	axis_init(
		object_name								:= CONCAT(prc_path, '_axis'), 
		axis_type								:= AXIS_TYPE_VIRTUAL, 
		encoder_scaling_factor					:= G_VIRTUAL_ENCODER_SCALING_FACTOR_DEGPINC,
		modulo									:= G_MODULO_360_DEG, 
		process									:= prc, 
		CONVERSION_this							:= axis);
	
	axis_set_max_dynamic(
		reference_velocity						:=	CONSTANTS.MAX_VELOCITY_MMpSEC,
		velocity								:=	CONSTANTS.MAX_VELOCITY_MMpSEC,
		acceleration							:=	CONSTANTS.MAX_ACCELERATION_MMpSEC2,
		deceleration							:=	CONSTANTS.MAX_DECELERATION_MMpSEC2,
		jerk									:=	CONSTANTS.MAX_JERK_MMpSEC3,
		following_error							:=	CONSTANTS.MAX_FOLLOWING_ERROR_MM,
		CONVERSION_this							:=	axis);

	jog_manager_add_axis(
		list_index					:= JOG_LIST_CSP_CASE_LOADER_VIRTUAL,
		axis						:= axis,
		master_axis					:= TRUE,
		jog_type					:= JOG_TYPE_ROTATIVE_PLUS,
		sw_limit_positive			:= 0.0,
		sw_limit_negative			:= 0.0,
		CONVERSION_this				:= csp_main_jogManager.jog_manager_virtual);
		
	boolean_init(
		object_name 							:= CONCAT(prc_path, '_case_loaded_bool'),
		process 								:= prc,
		CONVERSION_this							:= case_loaded_bool);

	check_section_asynchronous_mode_init(
		object_name:= CONCAT(prc_path, '_case_loaded_chksect'), 
		check_enable:=TRUE , 
		event_to_check:=CHECK_SECTION_EVENT_INPUT_ON , 
		execution_mode:=CHECK_SECTION_EXECUTION_WHEN_EVENT_OCCURRED , 
		diagnostic_enable:= FALSE , 
		status_bits_to_be_true:= common_global_variables.none, //ITEM_PRESENT, 
		status_bits_to_be_false:=common_global_variables.none, 
		_step_status_conditioning_execution:= FALSE, 
		status_bits_to_set:= ITEM_HAS_LOAD + ITEM_HAS_CARTON, 
		status_bits_to_reset:=common_global_variables.none , 
		reject_bit_to_set:= 0 , 
		_step:=26 , 
		first_step_to_write_offset:= 0, 
		number_of_steps_to_write:=1 , 
		reference_phase:=240 , 
		reference_phase_tolerance:= 0, 
		max_consecutive_failed_checks:= 1000000, 
		max_failed_checks_percentage:=10 , 
		products_for_failed_checks_percentage:= 10000000, 
		shift_register:= csp_case_main_statistics.sr, 
		process:= prc , 
		CONVERSION_this:= case_loaded_chksect);
		
	
			
	check_section_add_boolean_input(
			boolean_input:= case_loaded_bool,
			CONVERSION_this:= case_loaded_chksect);
		
		
	phase_init(
        object_name 				:= CONCAT(prc_path, '_load_check_ph'),
        phase 						:= 0,	//Set at runtime!
        delay 						:= 0,
        max_compensation 			:= 0,
        generator 					:= csp_main_motorization_virtualManager.phgen,
        process 					:= prc,
        CONVERSION_this 			:= load_check_ph);	
		
	phase_init(
        object_name 				:= CONCAT(prc_path, '_loader_run_check_ph'),
        phase 						:= 0,	//Set at runtime!
        delay 						:= 0,
        max_compensation 			:= 0,
        generator 					:= phgen, // CHANGE TO LOADER VIRTUAL PHGEN
        process 					:= prc,
        CONVERSION_this 			:= loader_run_check_ph);
		
	phase_generator_init(
		object_name					:= CONCAT(prc_path, '_phgen'), 
		modulo						:= axis_get_modulo(axis), 
		resolution					:= PHASE_GENERATOR_RESOLUTION_UNIT, 
		axis						:= axis, 
		process						:= prc, 
		CONVERSION_this				:= phgen);
		
		
	
	digital_check_and_message_init(
        object_name:= CONCAT(prc_path, 'product_load_failed_dchk'),
        alarm_if_input_off:= FALSE,
        alarm_delay:= 0,
        enabled_at_powerup:= TRUE,
        individual_reset:= FALSE,
        machine_reaction:=  MACHINE_REACTION_EMERGENCY_STOP,//MACHINE_REACTION_EMERGENCY_STOP,
        typology:=  MESSAGE_TYPOLOGY_ABNORMAL,//MESSAGE_TYPOLOGY_OBLIGATION,
        process:= prc,
        CONVERSION_this:= product_load_failed_dchk);
       
       
    digital_check_add_boolean(
        boolean:= product_load_failed,
        CONVERSION_this:= product_load_failed_dchk);	
		
	boolean_init(
		object_name 							:= CONCAT(prc_path, '_product_load_failed'),
		process 								:= prc,
		CONVERSION_this							:= product_load_failed);
		
		
	process_message_init(
		object_name					:=	CONCAT(prc_path, '_phase_faulted_aem'), 
		behaviour					:=	MESSAGE_BEHAVIOUR_EVENT,
		reset_timeout				:=	0,
		disableable					:=	TRUE,
		individual_reset			:=	FALSE,
		machine_reaction			:=	MACHINE_REACTION_NORMAL_STOP,
		typology					:=	MESSAGE_TYPOLOGY_ABNORMAL,
		process						:=	prc,
		CONVERSION_this				:=	phase_faulted_aem);
	
	timer_init(
		object_name					:= CONCAT(prc_path, 'phase_time_out_tmr'),
		process						:= prc,
		CONVERSION_this				:= phase_time_out_tmr);
		
	process_message_init(
		object_name					:=	CONCAT(prc_path, 'debug_immediate_stop_aem'), 
		behaviour					:=	MESSAGE_BEHAVIOUR_STATE,
		reset_timeout				:=	0,
		disableable					:=	TRUE,
		individual_reset			:=	FALSE,
		machine_reaction			:=	MACHINE_REACTION_NORMAL_STOP,
		typology					:=	MESSAGE_TYPOLOGY_ABNORMAL,
		process						:=	prc,
		CONVERSION_this				:=	debug_immediate_stop_aem);
		
	timer_init(
		object_name					:= CONCAT(prc_path, 'connection_time_out_tmr'),
		process						:= prc,
		CONVERSION_this				:= connection_time_out_tmr);
		
		
	process_message_init(
		object_name					:=	CONCAT(prc_path, '_connection_faulted_aem'), 
		behaviour					:=	MESSAGE_BEHAVIOUR_EVENT,
		reset_timeout				:=	0,
		disableable					:=	TRUE,
		individual_reset			:=	FALSE,
		machine_reaction			:=	MACHINE_REACTION_NORMAL_STOP,
		typology					:=	MESSAGE_TYPOLOGY_ABNORMAL,
		process						:=	prc,
		CONVERSION_this				:=	connection_faulted_aem);
		
	motorization_conditioner_init(
		object_name					:=	CONCAT(prc_path, 'connection_done_motcond'),
		velocity_limit				:=	0.0,
		velocity_limit_active		:=	FALSE,
		idle_handshake_active		:=	FALSE,
		execute_handshake_active	:=	TRUE,
		hold_handshake_active		:=	FALSE,
		suspend_handshake_active	:=	FALSE,
		complete_handshake_active	:=	FALSE,
		abort_handshake_active		:=	FALSE,
		stop_handshake_active		:=	FALSE,
		origin						:=	MOTORIZATION_CONDITIONER_ORIGIN_INTERNAL,
		manager						:=	csp_main_motorization_manager.motm,
		process						:=	prc,
		CONVERSION_this				:=	connection_done_motcond);
		
	process_message_init(
		object_name					:=	CONCAT(prc_path, '_Engagement_Error_aem'), 
		behaviour					:=	MESSAGE_BEHAVIOUR_EVENT,
		reset_timeout				:=	0,
		disableable					:=	TRUE,
		individual_reset			:=	FALSE,
		machine_reaction			:=	MACHINE_REACTION_EMERGENCY_STOP,
		typology					:=	MESSAGE_TYPOLOGY_ABNORMAL,
		process						:=	prc,
		CONVERSION_this				:=	Engagement_Error_aem);
		
END_IF

IF objects_running()
THEN
	motorization_conditioner_cycle(connection_done_motcond);
	phase_cycle(load_check_ph);
	phase_cycle(loader_run_check_ph);
	
	phase_generator_cycle(phgen);
	
	process_cycle(prc);
	axis_cycle(axis);
	
	digital_check_cycle(product_load_failed_dchk);
END_IF
END_ACTION

ACTION _read_process_image:
;
END_ACTION

ACTION _read_var_input:
disable_req := csp_case.disable_req;
;
END_ACTION

ACTION _set_runtime_properties:
(* Cam management *)
IF 	connection_done
THEN
	active_cam := axis.engaged_cam.cam_id;
END_IF
END_ACTION

ACTION _write_output:
;
END_ACTION

ACTION connection:
connection_conditions :=	
	NOT process_message_is_on(connection_faulted_aem)
	//AND
	//NOT jog_manager_is_jog_axis_active(JOG_LIST_CSP_CASE_VIRTUAL, csp_main_jogManager.jog_manager_virtual)
	AND
	phase_done;

(* connection_done reset *)
IF	connection_done
	AND	
	NOT connection_conditions
	AND
	NOT csp.o_machine_is_running
THEN
	connection_done := FALSE;
END_IF

(* Exit conditions *)
IF	NOT connection_conditions 
	AND
	NOT motorization_manager_is_stopping(csp_main_motorization_manager.motm)	
THEN	
	connection_status_next := CSP_CASE_STATUS_CONNECTION_ERROR;
	connection_status := connection_status_next;	
END_IF

(*************** MACHINE STATUS ***************)
CASE connection_status OF

	CSP_CASE_STATUS_CONNECTION_START:	(* Start connection *)
	
		IF	(
				motorization_manager_is_starting(csp_main_motorization_manager.motm) 
				OR
				jog_manager_is_jog_axis_active(JOG_LIST_CSP_CASE_VIRTUAL, csp_main_jogManager.jog_manager_virtual)
			)
		THEN
			connection_running := TRUE;
			connection_status_next := CSP_CASE_STATUS_CONNECTION_ENGAGE;
		END_IF
		
	CSP_CASE_STATUS_CONNECTION_ENGAGE:		
	
		master_offset_phase := csp_main_motorization_virtualManager.axis.actual_modulo_position;	
			
		axis_engage_cam(
			cam_id							:=	active_cam,	
			master_engage_mode				:=	AXIS_CAM_ENGAGE_RELATIVE,
			slave_engage_mode				:=	AXIS_CAM_ENGAGE_RELATIVE,
			activation_mode					:=	AXIS_CAM_ACTIVATION_IMMEDIATELY,
			activation_position				:=	0.0,
			master_scaling_mode				:=	AXIS_CAM_SCALING_MODE_USER_DEFINED,
			slave_scaling_mode				:=	AXIS_CAM_SCALING_MODE_AUTOOFFSET,
			master_offset					:=	LMOD(home_position_master_offset_deg + master_offset_phase, axis_get_modulo(csp_main_motorization_virtualManager.axis)),
			slave_offset					:=	0.0,
			master_scaling					:=	master_scaling,
			slave_scaling					:=	slave_scaling,
			interpolation_type				:=	AXIS_CAM_INTERPOLATION_SPLINE,	 
			master							:=	csp_main_motorization_virtualManager.axis,
			CONVERSION_this					:=	axis);
		
		connection_status_next:= CSP_TRANSFER_STATUS_CONNECTION_ENGAGED;
	
	CSP_CASE_STATUS_CONNECTION_ENGAGED:
	
		IF active_cam = 0
		THEN
			active_cam := next_cam;
		END_IF
	
		IF 	axis_is_cam_engaged(axis) 
		THEN				
			IF	active_cam <> next_cam
			THEN							
				connection_status_next := CSP_TRANSFER_STATUS_CONNECTION_CHANGE_CAM;
			ELSE
				connection_status_next:= CSP_TRANSFER_STATUS_CONNECTION_DONE;
			END_IF
		END_IF
		
	CSP_CASE_STATUS_CONNECTION_CHECK_CHANGE_CAM:						
		
		IF 	dwell
		THEN
			next_cam := DWELL_CAM;
			dwell:= FALSE;
		END_IF
				
		IF 	run
		THEN
			next_cam := FORWARD_CAM;
			run := FALSE;
		END_IF	
		
		IF	(active_cam <> next_cam)
			AND connection_conditions
		THEN							
			connection_status_next := CSP_TRANSFER_STATUS_CONNECTION_CHANGE_CAM;
		END_IF
			
		IF	NOT connection_motorization_moving
		THEN
			connection_status_next := CSP_TRANSFER_STATUS_CONNECTION_DONE;
		END_IF
			
	
	CSP_CASE_STATUS_CONNECTION_CHANGE_CAM:	
		engage_count := engage_count + 1;	
	
		axis_engage_cam(
			cam_id							:=	next_cam,	
			master_engage_mode				:=	AXIS_CAM_ENGAGE_ABSOLUTE,
			slave_engage_mode				:=	AXIS_CAM_ENGAGE_RELATIVE,
			activation_mode					:=	AXIS_CAM_ACTIVATION_NEXT_CYCLE,
			activation_position				:=	0,
			master_scaling_mode				:=	AXIS_CAM_SCALING_MODE_USER_DEFINED,
			slave_scaling_mode				:=	AXIS_CAM_SCALING_MODE_USER_DEFINED,
			master_offset					:=	home_position_master_offset_deg, 
			slave_offset					:=	0.0,
			master_scaling					:=	master_scaling,
			slave_scaling					:=	slave_scaling,
			interpolation_type				:=	AXIS_CAM_INTERPOLATION_SPLINE,	 
			master							:=	csp_main_motorization_virtualManager.axis,
			CONVERSION_this					:=	axis);	
	
		IF	motorization_manager_is_starting(csp_main_motorization_manager.motm)
		THEN
			connection_status_next := CSP_TRANSFER_STATUS_CONNECTION_DONE;
		ELSE
			IF 	axis_is_cam_engaged(axis)
			THEN
				connection_status_next := CSP_TRANSFER_STATUS_CONNECTION_WAIT_NEW_CAM;
			END_IF
		END_IF
	
	CSP_CASE_STATUS_CONNECTION_WAIT_NEW_CAM:
	
		IF	active_cam = next_cam
		THEN
			CASE next_cam OF
				DWELL_CAM:
					activation_position := next_activation_position;
				
				FORWARD_CAM:
					activation_position := 0;
					
			END_CASE
			connection_status_next := CSP_TRANSFER_STATUS_CONNECTION_CHECK_CHANGE_CAM;
		END_IF
		
		IF	NOT connection_motorization_moving
		THEN
			connection_status_next := CSP_TRANSFER_STATUS_CONNECTION_DONE;
		END_IF
		
	CSP_CASE_STATUS_CONNECTION_DONE:	(* Connection done *)	
	
		connection_running := FALSE;
		connection_done := TRUE;
		
		IF	motorization_manager_is_starting(csp_main_motorization_manager.motm)
		THEN
			motorization_conditioner_start_done(connection_done_motcond);							
			IF	active_cam <> next_cam
			THEN
				connection_status_next := CSP_TRANSFER_STATUS_CONNECTION_WAIT_NEW_CAM;
			ELSE
				connection_status_next := CSP_TRANSFER_STATUS_CONNECTION_CHECK_CHANGE_CAM;
			END_IF
		END_IF
	
	CSP_CASE_STATUS_CONNECTION_ERROR:	(* Connection error *)	
	
		IF 	connection_running
		THEN
			axis_disable(axis);
			connection_error := TRUE;						
		END_IF
		
		connection_running	:= FALSE;
		connection_done 	:= FALSE;	
		
		IF	connection_conditions
		THEN		
			connection_status_next := CSP_CASE_STATUS_CONNECTION_START;
		END_IF
		
END_CASE

IF 	NOT debug_state_machine
	OR
	debug_connection_machine_one_step	
THEN
	connection_status := connection_status_next;
	debug_connection_machine_one_step := FALSE;
END_IF

connection_motorization_moving	:= 
	motorization_manager_is_starting(csp_main_motorization_manager.motm)
	OR
	motorization_manager_is_execute(csp_main_motorization_manager.motm)
	OR
	motorization_manager_is_stopping(csp_main_motorization_manager.motm)
	OR
	motorization_manager_is_suspended(csp_main_motorization_manager.motm)
	OR
	motorization_manager_is_suspending(csp_main_motorization_manager.motm)
	OR
	motorization_manager_is_unsuspending(csp_main_motorization_manager.motm)
	OR 
	motorization_manager_is_holding(csp_main_motorization_manager.motm)
	OR
	motorization_manager_is_held(csp_main_motorization_manager.motm)
	OR
	motorization_manager_is_unholding(csp_main_motorization_manager.motm);	
	
(* Connection timeout *)
IF	(connection_running
	AND NOT debug_state_machine)	
	OR connection_error
THEN
	IF	timer_is_expired(connection_time_out_tmr)
	THEN
		process_message_set(1, connection_status, 0, connection_faulted_aem);
	END_IF
ELSE
	timer_restart(10000, connection_time_out_tmr);
END_IF
END_ACTION

ACTION phase:
phase_conditions :=
	axis_is_ok(FALSE, axis)
	AND
	process_is_ready(prc)
	AND
	process_subtree_is_ready(prc)
	//AND
	//NOT jog_manager_is_jog_axis_active(JOG_LIST_CSP_CASE_VIRTUAL, csp_main_jogManager.jog_manager_virtual)
	AND
	csp_main_motorization.motorization_axis_redefined_at_powerup
	AND
	NOT disable_req;		
	
(* phase_done reset *)
IF	phase_done
	AND
	NOT phase_conditions
	//AND 
	//NOT csp.o_machine_is_running
THEN
	//axis_disable(axis);
	phase_done:= FALSE;
END_IF

(* Exit condition *)
IF 	NOT phase_conditions
THEN
	phase_status_next := CSP_CASE_PHASE_STATUS_ERROR;
	phase_status := phase_status_next;	
END_IF

(*************** MACHINE STATUS ***************)
CASE phase_status OF

	CSP_CASE_PHASE_STATUS_START:	(* Start phasing *)
	
		IF	(
				motorization_manager_is_starting(csp_main_motorization_manager.motm) //TODOPZ: da decidere a che livello usare le variabili di i e o: wn_feeding.i_motorization_is_starting?					
				AND 
				loader_slaves_cammed
				//OR
				//jog_manager_is_jog_axis_active(JOG_LIST_CSP_CASE_VIRTUAL, csp_main_jogManager.jog_manager_virtual)
			)
		THEN
			phase_running := TRUE;			
			phase_status_next := CSP_CASE_PHASE_STATUS_DISABLE;
		END_IF
						
	CSP_CASE_PHASE_STATUS_DISABLE:
	
		axis_disable(axis);		
		
		IF 	axis_is_disabled(axis)
		THEN
			phase_status_next := CSP_CASE_PHASE_STATUS_ENABLE;
		END_IF
		
	CSP_CASE_PHASE_STATUS_ENABLE:
	
		axis_enable(axis);
		
		IF 	axis_is_enabled(axis)
		THEN
			phase_status_next := CSP_CASE_PHASE_STATUS_ENABLED;
		END_IF
		
	CSP_CASE_PHASE_STATUS_ENABLED:
	
		IF 	axis_is_standstill(axis) 
		THEN
			phase_status_next := CSP_CASE_PHASE_STATUS_CALCULATE_SLAVE_POSITION_REQUEST;								
		END_IF
		
	CSP_CASE_PHASE_STATUS_CALCULATE_SLAVE_POSITION_REQUEST:
	
		slave_position_has_been_calculated := FALSE;
	
		(* Gets the position of the master axis *)
		axis_calculate_cam_slave_master_position_deg := 
			LMOD(axis_get_actual_modulo_position(csp_main_motorization_virtualManager.axis)
			+ home_position_master_offset_deg, G_MODULO_360_DEG);
			
		(* Gets cam data for slave axis to master *)
		IF axis_calculate_cam_slave_dynamics_data(
			cam_id := active_cam,
			master_scaling := master_scaling,
			master_position := axis_calculate_cam_slave_master_position_deg,
			slave_scaling := slave_scaling,
			CONVERSION_this := axis)
		THEN
			phase_status_next := CSP_CASE_PHASE_STATUS_CALCULATING_SLAVE_POSITION;
		END_IF
	
	CSP_CASE_PHASE_STATUS_CALCULATING_SLAVE_POSITION:
	
		IF axis_cam_slave_dynamics_data_calculated(axis)
		THEN
			axis_calculated_cam_slave_position_deg := axis_get_cam_slave_dynamics_position(axis);
			slave_position_has_been_calculated := TRUE;
			phase_status_next := CSP_CASE_PHASE_STATUS_REQUEST;
				
		END_IF
		
	CSP_CASE_PHASE_STATUS_REQUEST:
		
		IF	axis_is_standstill(axis)
		THEN
			axis_move_absolute(
				position 		:= axis_calculated_cam_slave_position_deg,
				velocity 		:= phase_velocity_degps,
				direction		:= AXIS_SHORTEST_WAY,
				acceleration 	:= CONSTANTS.MOTOR_MAX_ACCELERATION_DEGPS2,
				deceleration 	:= CONSTANTS.MOTOR_MAX_DECELERATION_DEGPS2, 
				jerk 			:= CONSTANTS.MOTOR_MAX_JERK_DEGPS3, 
				buffer_mode 	:= AXIS_BUFFER_MODE_BUFFERED,
				CONVERSION_this := axis
				); 
			
		END_IF

		IF 	axis_is_absolute_moving(axis)
		THEN
			phase_status_next	:=	CSP_CASE_PHASE_STATUS_PHASING;
		END_IF

	CSP_CASE_PHASE_STATUS_PHASING:

		IF 	axis_is_standstill(axis)
		THEN
			phase_status_next	:=	CSP_TRANSFER_STATUS_PHASED;
		END_IF

	CSP_TRANSFER_STATUS_PHASED:

		IF 	engage_enable
		THEN
			phase_status_next := CSP_CASE_PHASE_STATUS_DONE;
		END_IF
		
		
	CSP_CASE_PHASE_STATUS_DONE:	(* Phase done *)	
		
		phase_running := FALSE;
		phase_done := TRUE;				
	
	CSP_CASE_PHASE_STATUS_ERROR:	(* Phase error *)
		

		IF	phase_running
		THEN
			phase_error := TRUE;
			axis_disable(axis);									
		END_IF
		phase_running := FALSE;
		
		IF	phase_conditions 	
		THEN
			phase_status_next := CSP_CASE_PHASE_STATUS_START;
		END_IF
		
END_CASE

IF 	NOT debug_state_machine
	OR
	debug_phase_machine_one_step	
THEN
	phase_status := phase_status_next;
	debug_phase_machine_one_step := FALSE;
END_IF

(* Phasing timeout *)
IF 	(phase_running
	AND NOT debug_state_machine)
	OR phase_error
THEN
	IF	timer_is_expired(phase_time_out_tmr)
	THEN
		process_message_set(1, phase_status, 0, phase_faulted_aem);
	END_IF
ELSE
	timer_restart(10000, phase_time_out_tmr);
END_IF
END_ACTION

END_PROGRAM

// ---- Application/CSP/Case/Transport/Virtual Master/csp_case_transport_virtualMaster.TcPOU
(*********************************** G.D S.p.A. - Technical Department ***********************************
============= PROGRAM INFO ============
FOLDER:             TBD
MACHINES INVOLVED:  TBD 

============= DESCRIPTION =============
csp machine declaration

============= REVISIONS ===============
Date		Version	 	Author      	Description             
----------	-------		------------  	--------------------------------------------
2019/04/05 	0000.00	 	M.Grasso		Creation of the PRG

**********************************************************************************************************)
(*$R process_ref := prc; $*)
PROGRAM csp_case_transport_virtualMaster
VAR
	
	prc:												process;
	prc_path:											STRING;
	test_pb:											BOOL:= FALSE;
	disable_pb:											BOOL:= FALSE;
	fsm_enable_condition:								BOOL := FALSE;
	fsm_next_status:									csp_case_transport_status_enum;
	fsm_status:											csp_case_transport_status_enum;
	phase_enable:										BOOL  := TRUE;
	axis: 												axis;
	phase_position_deg:									LREAL := 0;
	phase_velocity_degps:								LREAL := 20.0;
	axis_calculate_cam_slave_master_position_deg:		LREAL := 0.0;
	axis_calculated_cam_slave_position_deg:				LREAL := 0.0;
	axis_calculate_cam_master_slave_position_deg: 		LREAL := 0.0;
	axis_calculated_cam_master_position_deg: 			LREAL := 0.0;
	slave_position_has_been_calculated:					BOOL  := FALSE;
	master_position_has_been_calculated:				BOOL  := FALSE;
	engage_enable:										BOOL:=TRUE;
	target_position:									LREAL:=0;
	disable_req:										BOOL:=FALSE;
	debug_state_machine:								BOOL:=FALSE;
	debug_state_machine_one_step:						BOOL:=FALSE;
	os_minor_plow_phgen:								phase_generator;
	os_minor_plow_phwin:								phase_window;
	major_flap_phgen:									phase_generator;
	major_flap_phwin:									phase_window;
	
	transport_vm_phgen:									phase_generator;
	os_trailing_lug_pos:								LREAL;
	cam_id:												INT := LINEAR_CAM;
	slave_scaling_mm:									LREAL := 360; (*$P $*)
	master_scaling_deg:									LREAL := 360; (*$P $*)
	slave_scaling:										LREAL := 360; (*$P $*)
	master_scaling:										LREAL := 360; (*$P $*)
	home_position_master_offset_deg: 					LREAL := 0;
	running_cam:										BOOL;
	minor_plow_on: 										LREAL:=0; (*$P $*)
	minor_plow_off: 									LREAL:=100; (*$P $*)
	
	FLAG: 												STRING;
	transport_slaves_cammed:							BOOL:=FALSE;
	activation_position:    							LREAL:=0.001111;
	ls_flap_phgen:										phase_generator;
	ls_flap_on: 										LREAL := 110;
	ls_flap_off: 										LREAL := 125;
	ls_flap_phwin: 										phase_window;
	os_flap_phgen: 										phase_generator;
	os_flap_on: 										LREAL;
	os_flap_off: 										LREAL;
	os_flap_phwin: 										phase_window;
	debug: 												STRING;
	major_flap_check_on: 								LREAL:=352; (*$P $*)
	major_flap_check_off: 								LREAL:=357; (*$P $*)
	stop_for_reject: 									BOOL:=FALSE;
	PE_check: 											BOOL:=TRUE;	//initialized as true so transport virtual will run; toggle false to simulate case reject operation
	recovery_cycle:										BOOL:= FALSE;
	step_1: 											BOOL;
	step_2: 											BOOL;
	push_loader: 										BOOL;
	step_3: 											BOOL;
	step_4: 											BOOL;
	disengage_pos:										LREAL := 345;   
	latch: 												BOOL:= False;
	transport_request_latch: 							BOOL := FALSE;
	engage_after_estop: 								BOOL;
	Check_request_latch: 								BOOL := FALSE;
	Good_case_detected:									BOOL:= FALSE;
	Bad_case_detected:									BOOL:= FALSE;
	startup_follower_at_start_position:					BOOL:=FALSE;
	Startup_Good_case_detected:							BOOL := false;
	act_pos: 											LREAL := 0.995;
	reject_complete_test: 								BOOL := FALSE;
	test19:												BOOL := TRUE;
	
	PE_TEST: 											BOOL := TRUE;
	phase_done: 										BOOL := TRUE;
	Reject_again: 										BOOL := FALSE;
	pe_off: 											BOOL := TRUE;
	PE_Bypass_request:                                  BOOL:=FALSE;(*$P $*)
	consecutive_rejects_aem:							message;
	
	Abs_moved: 											BOOL;
	temp1: 												BOOL;

	Flap_control_engaged: 								BOOL;
	Reject_engaged: 									BOOL;
	Reject_disengaging: 								BOOL;
	Reject_disengaged: 									BOOL;
	Ready_to_collapse_bad_case: 						BOOL;
	Re_engaged_to_Case_Virtual: 						BOOL;
	detect_next_flaps: 									BOOL;(*$P desc:= DETECT START AND END PHASE OF FLAP EYES ON NEXT CASE; $*)
	eye_test_temp: 										BOOL;
	detected_start_phase: 								LREAL;(*$P desc:= DETECTED START PHASE OF FLAP EYES ON CASE; $*)
	detected_end_phase: 								LREAL;(*$P desc:= DETECTED END PHASE OF FLAP EYES ON CASE; $*)
	
	missing_os_fc_lower_pe_wem:							message;
	missing_os_fc_upper_pe_wem: 						message;
	missing_ls_fc_lower_pe_wem:							message;
	missing_ls_fc_upper_pe_wem: 						message;
	missing_flap: 										BOOL;
	transport_vm_ph: 									phase;
	Good_Case_For_SR: 									BOOLean;
	feed_chksect: 										check_section;
	boolean_is_resetting: 								BOOL;
	boolean_is_set: 									BOOL;
	reject_reset_boolean: 								BOOL;
	new_set: 											BOOL;
	axis_tolerance: 									INT := 30;
	phase_direction: 									BOOL;
END_VAR

VAR CONSTANT
	
	CONSTANTS:											csp_case_transport_constant_struct;

END_VAR
VAR_INPUT
	feed_reject_case_count: 							DINT;(*$M $*)
END_VAR

_read_var_input();

_object_manager();

IF NOT objects_running()
THEN
	RETURN;	
END_IF

_read_process_image();

_mode_manager();

CASE process_get_mode(prc) of
	MODE_ABSENT,
	MODE_INACTIVE:
		RETURN;
	MODE_TEST:
		_handle_process_test();
END_CASE

_set_runtime_properties();

(********************************* BODY *********************************)
				
IF  axis_is_cam_engaged(csp_case_transport_os_trailing.axis)
	AND axis_is_cam_engaged(csp_case_transport_os_leading.axis)
	AND axis_is_cam_engaged(csp_case_transport_ls_trailing.axis)
	AND axis_is_cam_engaged(csp_case_transport_ls_leading.axis)
	AND axis_is_cam_engaged(csp_case_tr_squaring_ls_leading.axis) 
	AND axis_is_cam_engaged(csp_case_tr_squaring_ls_trailing.axis)
	AND axis_is_cam_engaged(csp_case_tr_squaring_os_leading.axis)
	AND axis_is_cam_engaged(csp_case_tr_squaring_os_trailing.axis)
	AND axis_is_cam_engaged(csp_case_closing_os_horizontal.axis)
	AND axis_is_cam_engaged(csp_case_closing_os_upper.axis)
	AND axis_is_cam_engaged(csp_case_closing_os_lower.axis)
	AND axis_is_cam_engaged(csp_case_closing_ls_horizontal.axis)
	AND axis_is_cam_engaged(csp_case_closing_ls_upper.axis)
	AND axis_is_cam_engaged(csp_case_closing_ls_lower.axis)
	AND axis_is_cam_engaged(csp_case_discharge_speedbelt_ls.axis)
	AND axis_is_cam_engaged(csp_case_discharge_speedbelt_os.axis)
THEN
	transport_slaves_cammed := TRUE;
ELSE
	transport_slaves_cammed := FALSE;	
END_IF

IF axis_is_cam_engaged(csp_case_fc_os_lower_follower.axis)
	AND axis_is_cam_engaged(csp_case_fc_os_upper_follower.axis)
	AND axis_is_cam_engaged(csp_case_fc_os_lower_spreader.axis)
	AND axis_is_cam_engaged(csp_case_fc_os_upper_spreader.axis)
	AND axis_is_cam_engaged(csp_case_fc_ls_lower_follower.axis)
	AND axis_is_cam_engaged(csp_case_fc_ls_upper_follower.axis)
	AND axis_is_cam_engaged(csp_case_fc_ls_lower_spreader.axis)
	AND axis_is_cam_engaged(csp_case_fc_ls_upper_spreader.axis)
THEN
	Flap_control_engaged := TRUE;
ELSE
	Flap_control_engaged := FALSE;
END_IF



phase_window_set_phases_data(
	begin_phase:=  major_flap_check_on,
	end_phase:=  major_flap_check_off,
	begin_delay:= 0,
	end_delay:= 0,
	begin_max_compensation:= 0,
	end_max_compensation:= 0,
	CONVERSION_this:= major_flap_phwin);

IF	(
	digital_input_is_active(csp_case_fc_os_upper_sensors.flap_di)
	AND digital_input_is_active(csp_case_fc_os_lower_sensors.flap_di)
	AND digital_input_is_active(csp_case_fc_ls_upper_sensors.flap_di)
	AND digital_input_is_active(csp_case_fc_ls_lower_sensors.flap_di)
	AND NOT PE_Bypass_request
	)
	OR csp_case_main_services.dry_cycle_mode
	OR csp_main_jogManager.jog_is_active
THEN
	PE_check := TRUE;
ELSE
	Pe_check := FALSE;
END_IF

IF  ( phase_window_is_in_window(major_flap_phwin) OR (stop_for_reject AND (axis.actual_position > major_flap_check_on AND axis.actual_position < major_flap_check_off) AND axis_is_cam_engaged(axis) ))//phase_window_falling_edge(major_flap_phwin)/ 
	AND (csp_case_feed_arm_sensors.major_vacuum_sact.status = DIGITAL_ACTUATOR_STATUS_ACTIVATING OR digital_actuator_is_active(csp_case_feed_arm_sensors.major_vacuum_sact))
	AND (
		NOT PE_check
		OR NOT digital_input_is_active(csp_case_feed_arm_sensors.case_check_di)
		)
	AND csp_main_motorization_virtualManager.o_machine_is_moving 
	AND NOT csp_case_main_services.dry_cycle_mode
	AND NOT csp_case_feed_arm_sensors.mispicked_case 
THEN
	target_position := 358;
	stop_for_reject := TRUE;
	Bad_case_detected := TRUE;		
	boolean_reset(Good_Case_For_SR);
	boolean_is_resetting := TRUE;
	boolean_is_set := FALSE;
ELSIF (phase_window_is_in_window(major_flap_phwin) OR (stop_for_reject AND (axis.actual_position > major_flap_check_on AND axis.actual_position < major_flap_check_off) AND axis_is_cam_engaged(axis) ))//phase_window_falling_edge(major_flap_phwin)/ //AMR 9/1/2021
	AND PE_check
	AND (csp_case_feed_arm_sensors.major_vacuum_sact.status = DIGITAL_ACTUATOR_STATUS_ACTIVATING OR digital_actuator_is_active(csp_case_feed_arm_sensors.major_vacuum_sact))
	AND digital_input_is_active(csp_case_feed_arm_sensors.case_check_di)
	AND csp_main_motorization_virtualManager.o_machine_is_moving 
	OR csp_case_main_services.dry_cycle_mode
THEN
	boolean_set(Good_Case_For_SR);
	boolean_is_resetting := FALSE;
	boolean_is_set := TRUE;
END_IF

IF phase_edge(transport_vm_ph)//resetting at next index of shift register
THEN
	boolean_reset(Good_Case_For_SR);
END_IF

IF phase_window_falling_edge(major_flap_phwin)
	AND NOT PE_check
	AND digital_input_is_active(csp_case_feed_arm_sensors.case_check_di)
	AND NOT csp_case_main_services.dry_cycle_mode
THEN
	missing_flap := TRUE;
	ELSIF NOT digital_input_is_active(csp_case_fc_os_upper_sensors.flap_di)	AND missing_flap THEN
			process_message_set(1, 1, 1, missing_os_fc_upper_pe_wem); //message for missing fc os upper pe
	ELSIF NOT digital_input_is_active(csp_case_fc_os_lower_sensors.flap_di)	AND missing_flap THEN
			process_message_set(1, 1, 1, missing_os_fc_lower_pe_wem); //message for missing fc os lower pe
	ELSIF NOT digital_input_is_active(csp_case_fc_ls_upper_sensors.flap_di)	AND missing_flap 	THEN
			process_message_set(1, 1, 1, missing_ls_fc_upper_pe_wem); //message for missing fc ls upper pe
	ELSIF NOT digital_input_is_active(csp_case_fc_ls_lower_sensors.flap_di)	AND missing_flap 	THEN
			process_message_set(1, 1, 1, missing_ls_fc_lower_pe_wem); //message for missing fc ls lower pe
END_IF

IF(process_message_is_on(missing_os_fc_upper_pe_wem)
		OR process_message_is_on(missing_os_fc_lower_pe_wem)
		OR process_message_is_on(missing_ls_fc_upper_pe_wem)
		OR process_message_is_on(missing_ls_fc_lower_pe_wem))
		AND phase_edge(transport_vm_ph)
THEN
	process_message_reset(missing_os_fc_upper_pe_wem);
	process_message_reset(missing_os_fc_lower_pe_wem);
	process_message_reset(missing_ls_fc_upper_pe_wem);
	process_message_reset(missing_ls_fc_lower_pe_wem);
	missing_flap := FALSE;
END_IF

IF stop_for_reject
	AND csp_case_feed_virtualMaster.stop_during_reject
THEN
	stop_for_reject := FALSE;
END_IF

IF 	NOT csp_case_feed_virtualMaster.check_request
	AND csp_case_feed_virtualMaster.fsm_status <> CSP_CASE_FEED_STATUS_CAM_ENGAGED
THEN
	Bad_case_detected := FALSE;
	Good_case_detected := FALSE;
END_IF

IF csp_case_transport.transport_request 
THEN
	transport_request_latch := TRUE;
END_IF

IF transport_request_latch 
THEN
	IF axis.actual_modulo_position > 0 AND axis.actual_modulo_position < 5 OR stop_for_reject 
	THEN
		transport_request_latch := FALSE;
	END_IF
END_IF

IF 	csp_case_feed_virtualMaster.fsm_status = 157
THEN
	Startup_Good_case_detected := TRUE;
	startup_follower_at_start_position := TRUE;
ELSE
	Startup_Good_case_detected := FALSE;
	startup_follower_at_start_position := FALSE;	
END_IF

(* Turn on eye_test to capture the leading and trailing edge pe_check(when all flaps are opened successful). Use these values to then troubleshoot when eyes were lost or missed *)
IF 	detect_next_flaps
	AND NOT eye_test_temp
	AND pe_check
then
	detected_start_phase := csp_case_transport_virtualMaster.axis.actual_position;
	eye_test_temp := True;
	detect_next_flaps := False;
end_if

IF 	eye_test_temp
	AND NOT pe_check
then
	detected_end_phase := csp_case_transport_virtualMaster.axis.actual_position;
	eye_test_temp := False;
end_if

(* If stop occurs in reject operation, reset all reject bits to abort sequence and phase all axes back to starting to run *)
IF (
    machine_is_stop_emergency_active(csp.mch)
    OR machine_is_stop_normal_active(csp.mch)
    )
    AND STOP_FOR_REJECT
	OR csp_case_feed_virtualMaster.stop_during_reject
THEN
	Good_case_detected := FALSE;
	Check_request_latch :=FALSE;
	STOP_FOR_REJECT := FALSE;
	Check_request_latch :=FALSE;
	Bad_case_detected := FALSE;
	Reject_again := FALSE;
END_IF

IF (stop_for_reject 
	OR 
	reject_again)
	AND NOT temp1
THEN
	temp1 := TRUE;
	feed_reject_case_count := feed_reject_case_count + 1;
END_IF

IF 	NOT stop_for_reject 
	AND NOT reject_again
THEN
	temp1 := FALSE;
END_IF	

IF NOT csp_case_main_safety_emergency.sis.safely_closed_input.status 
	AND axis_is_cam_engaged(axis) 
THEN
	engage_after_estop := TRUE;
ELSIF csp_case_main_safety_emergency.sis.safely_closed_input.status 
	AND fsm_status = CSP_CASE_TRANSPORT_STATUS_CAM_ENGAGED 
THEN
	engage_after_estop := FALSE;
END_IF

fsm_enable_condition := axis_is_ok(FALSE, axis)
						AND
						process_is_ready(prc)
						AND
						NOT jog_manager_is_jog_axis_active(JOG_LIST_CSP_CASE_TRANSPORT_VIRTUAL, csp_main_jogManager.jog_manager_virtual)
						AND
						process_subtree_is_ready(prc)
						AND 
						NOT disable_req;
						
IF NOT fsm_enable_condition
	OR
	disable_req
	AND
	fsm_status <> CSP_CASE_TRANSPORT_STATUS_DISABLED
	AND
	fsm_status < CSP_CASE_TRANSPORT_STATUS_STOP_REQUEST
THEN
	fsm_status	:=	CSP_CASE_TRANSPORT_STATUS_STOP_REQUEST;	
END_IF

CASE fsm_status OF
	
	CSP_CASE_TRANSPORT_STATUS_NOT_INITIALIZED:
	
        IF	axis_is_ok(return_when_absent := TRUE, CONVERSION_this := axis)
        THEN
            fsm_next_status := CSP_CASE_TRANSPORT_STATUS_DISABLED;
        END_IF

		
	CSP_CASE_TRANSPORT_STATUS_DISABLED:

		IF	fsm_enable_condition
			AND
			(
				(motorization_manager_is_starting(csp_main_motorization_manager.motm))
				OR
				jog_manager_is_jog_axis_active(JOG_LIST_CSP_CASE_VIRTUAL, csp_main_jogManager.jog_manager_virtual)	
			)
		THEN
			boolean_reset(csp_case_feed_virtualMaster.case_feed_reject_active);
			fsm_next_status := CSP_CASE_TRANSPORT_STATUS_ENABLE_REQUEST;
		END_IF;

		
	CSP_CASE_TRANSPORT_STATUS_ENABLE_REQUEST:
	
		axis_enable(axis);
		IF axis_is_standstill(axis)
		THEN
	 			fsm_next_status	:=	CSP_CASE_TRANSPORT_STATUS_ENABLED;
		END_IF;		

		
	CSP_CASE_TRANSPORT_STATUS_ENABLED:


		fsm_next_status	:=	CSP_CASE_TRANSPORT_STATUS_HOME_REQUEST;

		
	CSP_CASE_TRANSPORT_STATUS_HOME_REQUEST: 

		fsm_next_status	:=	CSP_CASE_TRANSPORT_STATUS_HOME_DONE;

		
	CSP_CASE_TRANSPORT_STATUS_HOMING:

		axis.home.done := TRUE;
		IF axis_home_done(axis)
		THEN
			fsm_next_status	:=	CSP_CASE_TRANSPORT_STATUS_HOME_DONE;
		END_IF

		
	CSP_CASE_TRANSPORT_STATUS_HOME_DONE:
	
		IF phase_enable
		THEN
			fsm_next_status	:=	CSP_CASE_TRANSPORT_STATUS_CALCULATE_SLAVE_POSITION_REQUEST;
		END_IF
	
		
	CSP_CASE_TRANSPORT_STATUS_CALCULATE_SLAVE_POSITION_REQUEST:
	
		slave_position_has_been_calculated := FALSE;
		(* Gets the position of the master axis *)
		axis_calculate_cam_slave_master_position_deg := 
			LMOD(axis_get_actual_modulo_position(csp_case_virtualMaster.axis)
			+ home_position_master_offset_deg, G_MODULO_360_DEG);
		(* Gets cam data for slave axis to master *)
		IF axis_calculate_cam_slave_dynamics_data(
			cam_id := cam_id,
			master_scaling := master_scaling,
			master_position := axis_calculate_cam_slave_master_position_deg,
			slave_scaling := slave_scaling,
			CONVERSION_this := axis)
		THEN
				fsm_next_status := CSP_CASE_LOADER_STATUS_CALCULATING_SLAVE_POSITION;
		END_IF
		
		
	CSP_CASE_TRANSPORT_STATUS_CALCULATING_MASTER_POSITION:
	
		IF axis_cam_master_dynamics_data_calculated(csp_case_transport_os_trailing.axis)
		THEN
			axis_calculated_cam_master_position_deg := axis_get_cam_master_dynamics_master_axis_position_lower(axis);//csp_case_transport_os_trailing.axis
			master_position_has_been_calculated := TRUE;
			fsm_next_status := CSP_CASE_TRANSPORT_STATUS_PHASE_REQUEST;
		END_IF
		
		
	CSP_CASE_TRANSPORT_STATUS_CALCULATING_SLAVE_POSITION:
	
		IF axis_cam_slave_dynamics_data_calculated(axis)//csp_case_virtualMaster.axis
		THEN
			axis_calculated_cam_slave_position_deg := axis_get_cam_slave_dynamics_position(axis);
			slave_position_has_been_calculated := TRUE;
			fsm_next_status := CSP_CASE_TRANSPORT_STATUS_PHASE_REQUEST;
				
		END_IF
		
		
	CSP_CASE_TRANSPORT_STATUS_PHASE_REQUEST:

    	IF  LMOD((axis_calculated_cam_slave_position_deg + axis_tolerance+G_MODULO_360_DEG),G_MODULO_360_DEG)> LMOD((axis.actual_position + 360),G_MODULO_360_DEG)
        	OR
        	LMOD((axis_calculated_cam_slave_position_deg - axis_tolerance+G_MODULO_360_DEG),G_MODULO_360_DEG)< LMOD((axis.actual_position + 360),G_MODULO_360_DEG)
		THEN
			phase_direction := FALSE;    // shortest path
        ELSE
			phase_direction := TRUE; //forward
    	END_IF

		IF	axis_is_standstill(axis)(* Waits for slave axes to phase and cammed *)
			AND transport_slaves_cammed
		THEN			
			 axis_move_absolute(
				position 		:= axis_calculated_cam_slave_position_deg,
				velocity 		:= phase_velocity_degps,
				direction        := SEL(phase_direction, AXIS_SHORTEST_WAY, AXIS_POSITIVE_DIRECTION),//AXIS_SHORTEST_WAY,
				acceleration 	:= CONSTANTS.MAX_ACCELERATION_MMpSEC2/2,
				deceleration 	:= CONSTANTS.MAX_DECELERATION_MMpSEC2/2,
				jerk 			:= CONSTANTS.MAX_JERK_MMpSEC3/2, 
				buffer_mode 	:= AXIS_BUFFER_MODE_BUFFERED,
				CONVERSION_this 			:= axis
				); 
		END_IF

		IF axis_is_absolute_moving(axis)
		THEN
			fsm_next_status	:=	CSP_CASE_TRANSPORT_STATUS_PHASING;
		END_IF
	
	
	
	CSP_CASE_TRANSPORT_STATUS_PHASING:

		IF axis_is_standstill(axis)
		THEN
			phase_done := TRUE;
			fsm_next_status	:=	CSP_CASE_TRANSPORT_STATUS_PHASED;
		END_IF

		
	CSP_CASE_TRANSPORT_STATUS_PHASED:

		IF engage_enable	
		THEN
			fsm_next_status := CSP_CASE_TRANSPORT_STATUS_CAM_ENGAGED_REQ;
		END_IF


	CSP_CASE_TRANSPORT_STATUS_CAM_ENGAGED_REQ:
		 
		IF transport_slaves_cammed
		THEN	
			IF axis_get_command_velocity(csp_case_virtualMaster.axis) <1      
			THEN
				target_position :=0;
				axis_engage_cam(
					cam_id 				:= cam_id,
					master_engage_mode 	:= AXIS_CAM_ENGAGE_ABSOLUTE,
					slave_engage_mode 	:= AXIS_CAM_ENGAGE_ABSOLUTE, 
					activation_mode 	:= AXIS_CAM_ACTIVATION_IMMEDIATELY,
					activation_position	:= 0,
					master_scaling_mode	:= AXIS_CAM_SCALING_MODE_USER_DEFINED,
					slave_scaling_mode	:= AXIS_CAM_SCALING_MODE_USER_DEFINED,
					master_offset 		:= 0,
					slave_offset 		:= 0,
					master_scaling 		:= master_scaling,
					slave_scaling 		:= slave_scaling,
					interpolation_type 	:= AXIS_CAM_INTERPOLATION_SYSTEM_DEFAULT,
					master 				:= csp_case_virtualMaster.axis,
					CONVERSION_this 	:= axis);
			ELSE	
				axis_engage_cam(
					cam_id 				:= cam_id,
					master_engage_mode 	:= AXIS_CAM_ENGAGE_ABSOLUTE,
					slave_engage_mode 	:= AXIS_CAM_ENGAGE_ABSOLUTE, 
					activation_mode 	:= AXIS_CAM_ACTIVATION_AT_MASTER_CAM_POSITION,  
					activation_position	:= 0,
					master_scaling_mode	:= AXIS_CAM_SCALING_MODE_USER_DEFINED,
					slave_scaling_mode	:= AXIS_CAM_SCALING_MODE_USER_DEFINED,
					master_offset 		:= 0,
					slave_offset 		:= 0,
					master_scaling 		:= master_scaling,
					slave_scaling 		:= slave_scaling,
					interpolation_type 	:= AXIS_CAM_INTERPOLATION_SYSTEM_DEFAULT,
					master 				:= csp_case_virtualMaster.axis,
					CONVERSION_this 	:= axis);
			END_IF
		END_IF	
			
		IF	axis_is_cam_engaged(axis)
		THEN
	   		fsm_next_status := CSP_CASE_TRANSPORT_STATUS_CAM_ENGAGED;
		END_IF;
		
		
	CSP_CASE_TRANSPORT_STATUS_AXIS_ENGAGE_VERIFY :
	
		;
		
		
	CSP_CASE_TRANSPORT_STATUS_CAM_ENGAGED:
		
		IF 	NOT transport_request_latch 
			AND axis.actual_modulo_position > disengage_pos
		THEN
			fsm_next_status := CSP_CASE_TRANSPORT_STATUS_DISENGAGE_REQUEST;	
		END_IF
	
		IF NOT axis_is_enabled(axis)
		THEN
			fsm_next_status := CSP_CASE_TRANSPORT_STATUS_STOP_REQUEST;
		END_IF
	
		
	CSP_CASE_TRANSPORT_STATUS_RUNNING:

		IF motorization_manager_is_aborted(csp_main_motorization_manager.motm)
		THEN
			fsm_next_status := CSP_CASE_TRANSPORT_STATUS_STOP_REQUEST;
		END_IF
		
		
	CSP_CASE_TRANSPORT_STATUS_DISENGAGE_REQUEST:
	
		IF stop_for_reject 
		THEN
			target_position :=359.5; 
			fsm_next_status := CSP_CASE_TRANSPORT_STATUS_DISENGAGING;
		ELSE
			target_position :=0;
			fsm_next_status := CSP_CASE_TRANSPORT_STATUS_DISENGAGING;
		END_IF		
		
		
	CSP_CASE_TRANSPORT_STATUS_DISENGAGING:
	
	IF 	axis.actual_modulo_position >= disengage_pos 
		OR latch 
	THEN
		latch := TRUE;
		IF axis_disengage(
			mode:= AXIS_DISENGAGE_AND_ON_PHASE_STOP, 
			position:= target_position, 
			velocity:= 1000, 
			acceleration:= CONSTANTS.MAX_ACCELERATION_MMpSEC2, 
			deceleration:= CONSTANTS.MAX_DECELERATION_MMpSEC2, 
			jerk:= CONSTANTS.MAX_JERK_MMpSEC3, 
			CONVERSION_this:= axis)
		THEN
			IF  stop_for_reject 
			THEN
				latch := FALSE;				
				fsm_next_status := CSP_CASE_TRANSPORT_STATUS_REJECT_ABS_STEP_1;
			ELSE
				latch := FALSE;
				fsm_next_status := CSP_CASE_TRANSPORT_STATUS_CAM_ENGAGED_REQ;
			END_IF
		END_IF
	END_IF
	
	
	CSP_CASE_TRANSPORT_STATUS_STOP_REQUEST:

		axis_stop(
		    deceleration 	:= CONSTANTS.MAX_DECELERATION_MMpSEC2,
		    jerk 			:= CONSTANTS.MAX_JERK_MMpSEC3,
		    CONVERSION_this 			:= axis);

		IF 	axis_is_standstill(axis)
			OR
			NOT axis_is_ok(FALSE, axis)
			OR
			axis_is_disabled(axis)
		THEN
			fsm_next_status := CSP_CASE_TRANSPORT_STATUS_DISABLE_REQUEST;
		END_IF

		
	CSP_CASE_TRANSPORT_STATUS_DISABLE_REQUEST:
	
   		axis_disable(axis);
   		fsm_next_status := CSP_CASE_TRANSPORT_STATUS_DISABLING;

		
	CSP_CASE_TRANSPORT_STATUS_DISABLING:
	
        IF	axis_is_disabled(axis)
        THEN
            fsm_next_status := CSP_CASE_TRANSPORT_STATUS_DISABLED;
        END_IF;


	CSP_CASE_TRANSPORT_STATUS_REJECT_ABS_STEP_1:    //follower and spreaders move to zero
	
		Ready_to_collapse_bad_case := FALSE;
		
		IF stop_for_reject //AND csp_case_transport.flap_control_axes_standstill 
		THEN
			 reject_complete_test := FALSE;
			 Bad_case_detected := FALSE;
			 Reject_again := FALSE;
			 Check_request_latch := FALSE;
		END_IF
		
		IF axis_is_standstill(axis)
		THEN
			reject_complete_test := FALSE;
			Bad_case_detected := FALSE;
			Reject_again := FALSE;
			Check_request_latch := FALSE;
			axis_move_absolute(
				position 		:= csp_case_feed_virtualMaster.virtual_reject_disengage_position,
				velocity 		:= motorization_manager_get_nominal_velocity(csp_main_motorization_manager.motm),
				direction		:= AXIS_NEGATIVE_DIRECTION,
				acceleration 	:= csp_case_feed_virtualMaster.reject_accel,//CONSTANTS.MAX_ACCELERATION_MMpSEC2,
				deceleration 	:= csp_case_feed_virtualMaster.reject_accel,//CONSTANTS.MAX_DECELERATION_MMpSEC2,
				jerk 			:= CONSTANTS.MAX_JERK_MMpSEC3, 
				buffer_mode 	:= AXIS_BUFFER_MODE_BUFFERED,
				CONVERSION_this := axis); 
		END_IF
			
		IF 	axis_is_absolute_moving(axis)
		THEN
			fsm_next_status := CSP_CASE_TRANSPORT_STATUS_REJECT_ABS_STEP_2;
		END_IF
 
		
    CSP_CASE_TRANSPORT_STATUS_REJECT_ABS_STEP_2:    

		IF 	axis_is_standstill(axis) AND TRUNC(axis.actual_position) = 268
		THEN
			Ready_to_collapse_bad_case := TRUE;		
			fsm_next_status := CSP_CASE_TRANSPORT_STATUS_REJECT_ABS_STEP_3;
	 	END_IF
		
			 
	CSP_CASE_TRANSPORT_STATUS_REJECT_ABS_STEP_3:	
		
		IF csp_case_feed_virtualMaster.New_Case_Pick
		THEN	
			axis_engage_cam(
				cam_id 				:= cam_id,
				master_engage_mode 	:= AXIS_CAM_ENGAGE_ABSOLUTE,
				slave_engage_mode 	:= AXIS_CAM_ENGAGE_ABSOLUTE, 
				activation_mode 	:= AXIS_CAM_ACTIVATION_AT_MASTER_POSITION, 
				activation_position	:= csp_case_feed_virtualMaster.virtual_reject_disengage_position,
				master_scaling_mode	:= AXIS_CAM_SCALING_MODE_USER_DEFINED,
				slave_scaling_mode	:= AXIS_CAM_SCALING_MODE_AUTOOFFSET,
				master_offset 		:= 0,
				slave_offset 		:= 0,
				master_scaling 		:= master_scaling,
				slave_scaling 		:= slave_scaling,
				interpolation_type 	:= AXIS_CAM_INTERPOLATION_SYSTEM_DEFAULT,
				master 				:= csp_case_feed_virtualMaster.axis,
				CONVERSION_this 	:= axis);
		END_IF
			
		IF 	axis_is_cam_engaged(axis)
		THEN
			fsm_next_status := CSP_CASE_TRANSPORT_STATUS_REJECT_ABS_STEP_4;
		END_IF
		
		
	CSP_CASE_TRANSPORT_STATUS_REJECT_ABS_STEP_4:      

		 (* Determines if shift register will be set *)
		IF (axis.actual_position > major_flap_check_on AND axis.actual_position < major_flap_check_off) AND pe_check
			THEN 
				boolean_set(Good_Case_For_SR);
				new_set := TRUE;
		END_IF
		 
		IF 	axis_is_cam_engaged(axis) 
			AND	NOT pe_check  
			AND csp_case_feed_virtualMaster.follower_check_request							
		THEN
			Check_request_latch := FALSE;
			Bad_case_detected := TRUE;
			Reject_again := TRUE;
			process_message_set(1, 1, 1, consecutive_rejects_aem); //stop for consecutive reject 
		END_IF


        IF 	pe_check 
			AND axis_is_cam_engaged(axis)(*NOT bad_case_detected*) 
			AND csp_case_feed_virtualMaster.follower_check_request 
		THEN
			 Good_case_detected := TRUE;
			 Check_request_latch :=FALSE;
			 boolean_set(Good_Case_For_SR);
			 reject_reset_boolean := TRUE;
			 STOP_FOR_REJECT := FALSE;
			 Re_engaged_to_Case_Virtual := FALSE;
			 fsm_next_status := CSP_CASE_TRANSPORT_STATUS_RECOVERY_CAM_ENGAGED_REQ;
         END_IF
	
		
	CSP_CASE_TRANSPORT_STATUS_RECOVERY_CAM_ENGAGED_REQ:
		
		IF 	axis_is_cam_engaged(axis) 
			AND NOT Re_engaged_to_Case_Virtual
		THEN
			axis_disengage(
				mode:= AXIS_DISENGAGE_AND_STOP, 
				position 		:= 0,
				velocity:= 1000, 
				acceleration:= CONSTANTS.MAX_ACCELERATION_MMpSEC2, 
				deceleration:= CONSTANTS.MAX_DECELERATION_MMpSEC2, 
				jerk:= CONSTANTS.MAX_JERK_MMpSEC3, 
				CONVERSION_this 			:= axis ); 
			Reject_disengaging := TRUE;
		END_IF
		
		IF 	Reject_disengaging 
			AND axis_is_disengaged(axis)
		THEN
			Reject_disengaged := TRUE;
		END_IF
		

	IF 	csp_case_feed.feed_request
		AND axis_is_standstill(axis)
		AND TRUNC(axis.actual_position) = 0
		AND Reject_disengaged
	THEN
		
		axis_engage_cam(
				cam_id 				:= cam_id,
				master_engage_mode 	:= AXIS_CAM_ENGAGE_ABSOLUTE,
				slave_engage_mode 	:= AXIS_CAM_ENGAGE_ABSOLUTE, 
				activation_mode 	:= AXIS_CAM_ACTIVATION_IMMEDIATELY, 
				activation_position	:= 0,
				master_scaling_mode	:= AXIS_CAM_SCALING_MODE_USER_DEFINED,
				slave_scaling_mode	:= AXIS_CAM_SCALING_MODE_USER_DEFINED,
				master_offset 		:= 0,
				slave_offset 		:= 0,
				master_scaling 		:= master_scaling,
				slave_scaling 		:= slave_scaling,
				interpolation_type 	:= AXIS_CAM_INTERPOLATION_SYSTEM_DEFAULT,
				master 				:= csp_case_virtualMaster.axis,
				CONVERSION_this 	:= axis);	
		Re_engaged_to_Case_Virtual := TRUE;
	END_IF			
		
	IF 	axis_is_cam_engaged(axis) 
		AND Re_engaged_to_Case_Virtual 
	THEN
		step_4:= FALSE;
		Abs_moved := FALSE; //Resets bit for reject again
		reject_complete_test := TRUE;
		Good_case_detected := FALSE;
		Reject_disengaged := FALSE;
		Reject_disengaging := FALSE;
		fsm_next_status := CSP_CASE_TRANSPORT_STATUS_CAM_ENGAGED;
	
		IF pe_check (*NOT bad_case_detected*) 
			AND Stop_for_reject
			AND axis_is_cam_engaged(csp_case_fc_os_lower_follower.axis)
			AND axis_is_cam_engaged(csp_case_fc_os_upper_follower.axis)
			AND axis_is_cam_engaged(csp_case_fc_ls_lower_follower.axis)
			AND axis_is_cam_engaged(csp_case_fc_ls_upper_follower.axis)
			AND csp_case_transport.Spreaders_Extended
			AND axis_is_cam_engaged(csp_case_feed_virtualMaster.axis)	
		THEN
			STOP_FOR_REJECT := FALSE;
		END_IF
	END_IF
		
END_CASE;

IF NOT debug_state_machine
	OR
	debug_state_machine_one_step
THEN
	fsm_status := fsm_next_status;
	debug_state_machine_one_step := FALSE;
END_IF

(************************************************************************)

_handle_messages();

_write_output();

ACTION _handle_messages:
IF (
	machine_is_stopped(csp.mch)
	OR machine_is_stop_emergency_active(csp.mch)
	)
	AND process_message_is_on(consecutive_rejects_aem)
THEN
	bad_case_detected := FALSE;
	Good_case_detected := FALSE;
	process_message_reset(consecutive_rejects_aem);
		
END_IF;
END_ACTION

ACTION _handle_process_test:
;
END_ACTION

ACTION _mode_manager:
IF process_mode_req_is_pending(prc)
THEN
    process_apply_mode_req_first_step(prc);
    CASE process_get_mode(prc) OF
        MODE_TO_ABSENT:
			;
        MODE_TO_INACTIVE:
			;
        MODE_TO_TEST:
			;
        MODE_TO_OPERATIONAL:
			;
    END_CASE
    process_apply_mode_req_second_step(prc);
END_IF
END_ACTION

ACTION _object_manager:
IF objects_initialization()
THEN
	sub_process_init(
		object_name								:= 'csp_case_transport_virtualMaster.prc', 
		process									:= csp_case_transport.prc, 
		CONVERSION_this							:= prc);
		
	prc_path 									:= process_get_path(prc);
	
	axis_init(
		object_name								:= CONCAT(prc_path, '_axis'), 
		axis_type								:= AXIS_TYPE_VIRTUAL, 
		encoder_scaling_factor					:= G_VIRTUAL_ENCODER_SCALING_FACTOR_DEGPINC,
		modulo									:= G_MODULO_360_DEG, 
		process									:= prc, 
		CONVERSION_this							:= axis);
	
	axis_set_max_dynamic(
		reference_velocity						:=	CONSTANTS.MAX_VELOCITY_MMpSEC,
		velocity								:=	CONSTANTS.MAX_VELOCITY_MMpSEC,
		acceleration							:=	CONSTANTS.MAX_ACCELERATION_MMpSEC2,
		deceleration							:=	CONSTANTS.MAX_DECELERATION_MMpSEC2,
		jerk									:=	CONSTANTS.MAX_JERK_MMpSEC3,
		following_error							:=	CONSTANTS.MAX_FOLLOWING_ERROR_MM,
		CONVERSION_this							:=	axis);
		
	jog_manager_add_axis(
		list_index								:= JOG_LIST_CSP_CASE_TRANSPORT_VIRTUAL,
		axis									:= axis,
		master_axis								:= TRUE,
		jog_type								:= JOG_TYPE_ROTATIVE_PLUS,
		sw_limit_positive						:= 0.0,
		sw_limit_negative						:= 0.0,
		CONVERSION_this							:= csp_main_jogManager.jog_manager_virtual);

//Created to be the axis for the shift registers	
	phase_generator_init(
		object_name								:=CONCAT(PRC_PATH, '_transport_vm_phgen'), 
		modulo									:=360 , 
		resolution								:= PHASE_GENERATOR_RESOLUTION_UNIT, 
		axis									:=axis, 
		process									:=prc , 
		CONVERSION_this							:= transport_vm_phgen);
//Upper major flap check cam and phase generator	

//Lower major flap check cam and phase generator		
	
	phase_window_init(
		object_name								:=CONCAT(PRC_PATH, '_major_lower_flap_phwin'), 
		begin_phase								:=major_flap_check_on, 
		end_phase								:=major_flap_check_off, 
		begin_delay								:=0, 
		end_delay								:=0, 
		begin_max_compensation					:=0, 
		end_max_compensation					:=0, 
		generator								:=transport_vm_phgen , 
		process									:=prc , 
		CONVERSION_this							:=major_flap_phwin);	

//OS minor plow cam window and phase generator
	
	phase_window_init(
		object_name								:=CONCAT(PRC_PATH, '_os_minor_plow_phwin'), 
		begin_phase								:=minor_plow_on, 
		end_phase								:=minor_plow_off, 
		begin_delay								:=0, 
		end_delay								:=0, 
		begin_max_compensation					:=0, 
		end_max_compensation					:=0, 
		generator								:=transport_vm_phgen , 
		process									:=prc , 
		CONVERSION_this							:=os_minor_plow_phwin);	



//LS open flap cam window and phase generator
	
	
	phase_window_init(
		object_name								:=CONCAT(PRC_PATH, '_ls_flap_phwin'), 
		begin_phase								:=ls_flap_on, 
		end_phase								:=ls_flap_off, 
		begin_delay								:=0, 
		end_delay								:=0, 
		begin_max_compensation					:=0, 
		end_max_compensation					:=0, 
		generator								:=transport_vm_phgen , 
		process									:=prc , 
		CONVERSION_this							:=ls_flap_phwin);	

//OS open flap cam window and phase generator		
	
	phase_window_init(
		object_name								:=CONCAT(PRC_PATH, '_os_flap_phwin'), 
		begin_phase								:=os_flap_on, 
		end_phase								:=os_flap_off, 
		begin_delay								:=0, 
		end_delay								:=0, 
		begin_max_compensation					:=0, 
		end_max_compensation					:=0, 
		generator								:=transport_vm_phgen , 
		process									:=prc , 
		CONVERSION_this							:=os_flap_phwin);
		
//transport vm phase edge		
	 phase_init(
        object_name               				:= CONCAT(prc_path, '_transport_vm_ph'),
        phase                         			:= 0,    //Set at runtime!
        delay                         			:= 0,
        max_compensation             			:= 0,
        generator                    			:= transport_vm_phgen, 
        process                     			:= prc,
        CONVERSION_this             			:= transport_vm_ph);

		
		process_message_init(
		object_name:= CONCAT(prc_path, '_consecutive_reject_aem'), 
		behaviour:= MESSAGE_BEHAVIOUR_STATE, 
		reset_timeout:= 0, 
		disableable:= FALSE, 
		individual_reset:= FALSE, 
		machine_reaction:= MACHINE_REACTION_STOP_IN_PHASE_ONE, 
		typology:= MESSAGE_TYPOLOGY_ABNORMAL, 
		process:= prc, 
		CONVERSION_this:= consecutive_rejects_aem);
		
		process_message_init(
        object_name:= CONCAT(prc_path, '_missing_os_fc_lower_pe_wem'),
        behaviour:= MESSAGE_BEHAVIOUR_EVENT,
        reset_timeout:= 0,
        disableable:= TRUE,
        individual_reset:= FALSE,
        machine_reaction:= MACHINE_REACTION_NO_STOP,
        typology:=  MESSAGE_TYPOLOGY_NORMAL,
        process:= prc,
        CONVERSION_this:= missing_os_fc_lower_pe_wem);       
       
       
        process_message_init(
        object_name:= CONCAT(prc_path, '_missing_os_fc_upper_pe_wem'),
        behaviour:= MESSAGE_BEHAVIOUR_EVENT,
        reset_timeout:= 0,
        disableable:= TRUE,
        individual_reset:= FALSE,
        machine_reaction:= MACHINE_REACTION_NO_STOP,
        typology:=  MESSAGE_TYPOLOGY_NORMAL,
        process:= prc,
        CONVERSION_this:= missing_os_fc_upper_pe_wem);       
       
        process_message_init(
        object_name:= CONCAT(prc_path, '_missing_ls_fc_lower_pe_wem'),
        behaviour:= MESSAGE_BEHAVIOUR_EVENT,
        reset_timeout:= 0,
        disableable:= TRUE,
        individual_reset:= FALSE,
        machine_reaction:= MACHINE_REACTION_NO_STOP,
        typology:=  MESSAGE_TYPOLOGY_NORMAL,
        process:= prc,
        CONVERSION_this:= missing_ls_fc_lower_pe_wem);       
       
       
        process_message_init(
        object_name:= CONCAT(prc_path, '_missing_ls_fc_upper_pe_wem'),
        behaviour:= MESSAGE_BEHAVIOUR_EVENT,
        reset_timeout:= 0,
        disableable:= TRUE,
        individual_reset:= FALSE,
        machine_reaction:= MACHINE_REACTION_NO_STOP,
        typology:=  MESSAGE_TYPOLOGY_NORMAL,
        process:= prc,
        CONVERSION_this:= missing_ls_fc_upper_pe_wem);       

	boolean_init(
		object_name					:= CONCAT(prc_path, '_Good_Case_For_SR'), 
		process						:= prc, 
		CONVERSION_this				:= Good_Case_For_SR);		
		
		//AMR 9/1/2021
	check_section_phase_mode_init(
		object_name								:= CONCAT(prc_path, '_feed_chksect'), 
		check_enable							:= TRUE, 
		event_to_check							:= CHECK_SECTION_EVENT_INPUT_ON, 
		execution_mode							:= CHECK_SECTION_EXECUTION_WHEN_EVENT_OCCURRED, 
		diagnostic_enable						:= FALSE, 
		status_bits_to_be_true					:= common_global_variables.NONE, 
		status_bits_to_be_false					:= common_global_variables.NONE, 
		_step_status_conditioning_execution		:= FALSE, 
		status_bits_to_set						:= ITEM_CASE_FEED + ITEM_HAS_LS_LOWER_FLAP + ITEM_HAS_LS_UPPER_FLAP + ITEM_HAS_OS_UPPER_FLAP + ITEM_HAS_OS_LOWER_FLAP, //+ ITEM_CASE_FEED,  
		status_bits_to_reset					:= common_global_variables.NONE, 
		reject_bit_to_set						:= 0, 
		_step									:= 25, 
		first_step_to_write_offset				:= 0, 
		number_of_steps_to_write				:= 1, 
		check_phase								:= 359, 
		max_consecutive_failed_checks			:= 0, 
		max_failed_checks_percentage			:= 0, 
		products_for_failed_checks_percentage	:= 0, 
		shift_register							:= csp_case_main_statistics.sr , 
		process									:= prc, 
		CONVERSION_this							:= feed_chksect);
		
	check_section_add_boolean_input(
		boolean_input:= Good_Case_For_SR, 
		CONVERSION_this:= feed_chksect);	
END_IF

IF objects_running()
THEN
	process_cycle(prc);
	axis_cycle(axis);
	
	phase_generator_cycle(transport_vm_phgen);
	phase_window_cycle(major_flap_phwin);
	phase_cycle(transport_vm_ph);	
	phase_window_cycle(os_minor_plow_phwin);
	phase_window_cycle(os_flap_phwin);
	phase_window_cycle(ls_flap_phwin);
	
END_IF
END_ACTION

ACTION _read_process_image:
;
END_ACTION

ACTION _read_var_input:
disable_req := csp_case.disable_req;
;
END_ACTION

ACTION _set_runtime_properties:

END_ACTION

ACTION _write_output:
;
END_ACTION

END_PROGRAM

// ---- Application/CSP/Main/Jog Manager/csp_main_jogManager.TcPOU
(*********************************** G.D S.p.A. - Technical Department ***********************************
============= PROGRAM INFO ============
FOLDER:             TBD
MACHINES INVOLVED:  TBD 

============= DESCRIPTION =============

============= REVISIONS ===============
Date		Version	 	Author      	Description             
----------	-------		------------  	--------------------------------------------
2020/05/18 	0000.00	 	Infomotion srl	Creation of the PRG

**********************************************************************************************************)
(*$R
	process_ref := prc;
$*)
PROGRAM csp_main_jogManager
VAR
	prc:						process;
	prc_path:					STRING;
	AccDec_divider:				INT:=10;
	
	jog_activation_condition:	BOOL;
	jog_manager_real:			jog_manager;	
	jog_list_real:				csp_jog_list_real;			(*$P desc := jog real axis selection list; $*)
	jog_list_real_pow:			parameter_overwrite;
	jog_manager_virtual:		jog_manager;
	jog_list_virtual:			csp_jog_list_virtual;		(*$P desc := jog virtual axis selection list; $*)
	jog_list_virtual_pow:		parameter_overwrite;
	jog_manager_accuchange:		jog_manager;	
	jog_list_accuchange:		csp_jog_list_AccUChange;	(*$P desc := jog Acc-U-Change axis selection list; $*)
	jog_list_accuchange_pow:	parameter_overwrite;		
	
	jog_is_active:				BOOL;
	jog_is_active_wem:	 		message;
	
	di_pendant_positive:		digital_input;
	pendant_positive_cmd:		BOOL;
	di_pendant_negative:		digital_input;
	pendant_negative_cmd:		BOOL;
	
	first_loop:					BOOL := TRUE;
		
	debug_active:				BOOL := FALSE;
	debug_pendant_positive:		BOOL := FALSE;
	debug_pendant_negative:		BOOL := FALSE;
	
	accu_speeds:				csp_jog_accu_suggested_speeds;
	accu_axis_suggested_speed:	LREAL;	(*$M $*)
	prev_accu_axis_selected:	UINT := 0;
	
END_VAR

_read_var_input();

_objects_manager();

IF 	NOT objects_running()
THEN
	RETURN;
END_IF

_read_process_image();

_mode_manager();

CASE process_get_mode (CONVERSION_this := prc) OF

	MODE_ABSENT,
	MODE_INACTIVE:
		RETURN;

	MODE_TEST:
		_handle_process_test();
END_CASE

_set_runtime_properties();

(********************************* BODY *********************************)
	
IF 	first_loop
THEN
	parameter_overwrite_set_enum_value(JOG_LIST_NO_RAXIS_SELECT_TO_JOG, jog_list_real_pow);
	parameter_overwrite_set_enum_value(JOG_LIST_NO_VAXIS_SELECT_TO_JOG, jog_list_virtual_pow);
	parameter_overwrite_set_enum_value(JOG_LIST_NO_UAXIS_SELECT_TO_JOG, jog_list_accuchange_pow);			
END_IF
first_loop := FALSE;

jog_activation_condition :=
					NOT
					(
						motorization_manager_is_starting(csp_main_motorization_manager.motm)
						OR
						motorization_manager_is_execute(csp_main_motorization_manager.motm)
						OR
						motorization_manager_is_stopping(csp_main_motorization_manager.motm)
					);
					
jog_manager_set_jog_activation_condition(
	jog_activation_condition	:= jog_activation_condition,								
	CONVERSION_this				:= jog_manager_real);
jog_manager_set_jog_activation_condition(
	jog_activation_condition	:= jog_activation_condition,								
	CONVERSION_this				:= jog_manager_virtual);
jog_manager_set_jog_activation_condition(
	jog_activation_condition	:= jog_activation_condition,								
	CONVERSION_this				:= jog_manager_accuchange);

IF jog_list_real <> JOG_LIST_NO_RAXIS_SELECT_TO_JOG
THEN
	jog_manager_set_list_selected(
		list_selected		:= jog_list_real,
		CONVERSION_this		:= jog_manager_real);
END_IF

IF jog_list_virtual <> JOG_LIST_NO_VAXIS_SELECT_TO_JOG
THEN
	jog_manager_set_list_selected(
		list_selected		:= jog_list_virtual,
		CONVERSION_this		:= jog_manager_virtual);
END_IF

IF jog_list_accuchange <> JOG_LIST_NO_UAXIS_SELECT_TO_JOG
THEN
	jog_manager_set_list_selected(
		list_selected		:= jog_list_accuchange,
		CONVERSION_this		:= jog_manager_accuchange);
END_IF
	
jog_is_active :=
	(jog_manager_is_jog_active(jog_manager_real) AND jog_list_real <> JOG_LIST_NO_RAXIS_SELECT_TO_JOG)
	OR
	(jog_manager_is_jog_active(jog_manager_virtual) AND jog_list_virtual <> JOG_LIST_NO_VAXIS_SELECT_TO_JOG)
	OR
	(jog_manager_is_jog_active(jog_manager_accuchange) AND jog_list_accuchange <> JOG_LIST_NO_UAXIS_SELECT_TO_JOG); 
	

accu_axis_suggested_speed := accu_speeds.Suggested_Speeds[jog_manager_accuchange.CONVERSION_private.list_selected];	

IF jog_manager_accuchange.CONVERSION_private.list_selected <> prev_accu_axis_selected
THEN
	jog_manager_accuchange.axis_speed_linear := accu_axis_suggested_speed;
END_IF
prev_accu_axis_selected := jog_manager_accuchange.CONVERSION_private.list_selected;

IF	csp_main.o_reset_button
THEN
	jog_manager_stop_jog_absolute_movement(jog_manager_real);
	jog_manager_stop_jog_absolute_movement(jog_manager_virtual);
	jog_manager_stop_jog_absolute_movement(jog_manager_accuchange);	
END_IF

(************************************************************************)

_handle_messages();

_write_output();

ACTION _handle_messages:
IF	jog_is_active
THEN
	process_message_set(0, 0, 0, jog_is_active_wem);
ELSE	
	process_message_reset(jog_is_active_wem);
END_IF
END_ACTION

ACTION _handle_process_test:
;
END_ACTION

ACTION _mode_manager:
IF process_mode_req_is_pending(CONVERSION_this := prc)
THEN
    process_apply_mode_req_first_step(CONVERSION_this := prc);
    CASE process_get_mode(CONVERSION_this := prc) OF
        MODE_TO_ABSENT:
            ;
        MODE_TO_INACTIVE:
            ;
        MODE_TO_TEST:
            ;
        MODE_TO_OPERATIONAL:
            ;
    END_CASE
    process_apply_mode_req_second_step(CONVERSION_this := prc);
END_IF;
END_ACTION

ACTION _objects_manager:
IF objects_initialization()
THEN
    sub_process_init(
	    object_name 		:= 'csp_main_jogManager.prc',
        process				:= csp_main.prc,
        CONVERSION_this		:= prc);

	prc_path 				:= process_get_path(prc);
	
	(*Jog manager initialization*)
	jog_manager_init(
		object_name 		:= CONCAT(prc_path, '_jog_manager_real'),
		process				:= prc,
		CONVERSION_this		:= jog_manager_real);
		
	jog_manager_add_parent(
		parent				:= jog_manager_virtual,
		CONVERSION_this		:= jog_manager_real);
	
	jog_manager_add_parent(
		parent				:= jog_manager_accuchange,
		CONVERSION_this		:= jog_manager_real);
	
		
	jog_manager_init(
		object_name 		:= CONCAT(prc_path, '_jog_manager_virtual'),
		process				:= prc,
		CONVERSION_this		:= jog_manager_virtual);
		
	jog_manager_add_parent(
		parent				:= jog_manager_real,
		CONVERSION_this		:= jog_manager_virtual);
	
	jog_manager_add_parent(
		parent				:= jog_manager_accuchange,
		CONVERSION_this		:= jog_manager_virtual);
	
		
	jog_manager_init(
		object_name 		:= CONCAT(prc_path, '_jog_manager_accuchange'),
		process				:= prc,
		CONVERSION_this		:= jog_manager_accuchange);
	
	jog_manager_add_parent(
		parent				:= jog_manager_real,
		CONVERSION_this		:= jog_manager_accuchange);
	
	jog_manager_add_parent(
		parent				:= jog_manager_virtual,
		CONVERSION_this		:= jog_manager_accuchange);
		
	(*Pendant initialization*)
	digital_input_init(
		object_name 		:= CONCAT(prc_path, '_di_pendant_positive'),
		polarity_direct		:= TRUE,
		process				:= prc,
		CONVERSION_this		:= di_pendant_positive);

	digital_input_init(
		object_name 		:= CONCAT(prc_path, '_di_pendant_negative'),
		polarity_direct		:= TRUE,
		process				:= prc,
		CONVERSION_this		:= di_pendant_negative);
	
	jog_manager_add_pendant(
		di_pendant_positive	:= di_pendant_positive,
		di_pendant_negative	:= di_pendant_negative,
		CONVERSION_this		:= jog_manager_real);
	
	jog_manager_add_shared_pendant(
		parent				:= jog_manager_real,
		CONVERSION_this		:= jog_manager_virtual);
	
	jog_manager_add_shared_pendant(
		parent				:= jog_manager_real,
		CONVERSION_this		:= jog_manager_accuchange);
		
	(*Parameter overwrite and alarm initialization*)	
	parameter_overwrite_enum_init(
		object_name 		:= CONCAT(prc_path, '_jog_list_real_pow'),
		adr_of_parameter	:= ADR(jog_list_real),
		process				:= prc,
		CONVERSION_this		:= jog_list_real_pow);
	
	parameter_overwrite_enum_init(
		object_name 		:= CONCAT(prc_path, '_jog_list_virtual_pow'),
		adr_of_parameter	:= ADR(jog_list_virtual),
		process				:= prc,
		CONVERSION_this		:= jog_list_virtual_pow);
		
	parameter_overwrite_enum_init(
		object_name 		:= CONCAT(prc_path, '_jog_list_accuchange_pow'),
		adr_of_parameter	:= ADR(jog_list_accuchange),
		process				:= prc,
		CONVERSION_this		:= jog_list_accuchange_pow);
	
	process_message_init(
		object_name			:=	CONCAT(prc_path, '_jog_is_active_wem'), 
		behaviour			:=	MESSAGE_BEHAVIOUR_STATE,
		reset_timeout		:=	0,
		disableable			:=	TRUE,
		individual_reset	:=	FALSE,
		machine_reaction	:=	MACHINE_REACTION_NO_STOP,
		typology			:=	MESSAGE_TYPOLOGY_OBLIGATION,
		process				:=	prc,
		CONVERSION_this		:=	jog_is_active_wem);
END_IF

IF objects_running()
THEN
	process_cycle(prc);	
	
	jog_manager_cycle(jog_manager_real);
	jog_manager_cycle(jog_manager_virtual);
	jog_manager_cycle(jog_manager_accuchange);
END_IF
END_ACTION

ACTION _read_process_image:
;
END_ACTION

ACTION _read_var_input:
IF	debug_active
THEN
	IF	debug_pendant_positive
		AND
		pendant_negative_cmd
	THEN
		debug_pendant_negative := FALSE;		
	END_IF
	
	IF	debug_pendant_negative
		AND
		pendant_positive_cmd
	THEN
		debug_pendant_positive := FALSE;		
	END_IF
	
	di_pendant_positive.field.status := debug_pendant_positive;
	di_pendant_negative.field.status := debug_pendant_negative;
END_IF

digital_input_read(pendant_positive_cmd, di_pendant_positive);
digital_input_read(pendant_negative_cmd, di_pendant_negative);
END_ACTION

ACTION _set_runtime_properties:
;
END_ACTION

ACTION _write_output:
;
END_ACTION

END_PROGRAM

// ---- POUs/AFL extensions/jog_manager/commands/jog_manager_set_jog_activation_condition.TcPOU
(*$
	Set the jog activation condition in <b><i>this</i></b>.
	The method returns <i>TRUE</i> if the command is accepted, otherwise it returns <i>FALSE</i>.
$*)
FUNCTION jog_manager_set_jog_activation_condition : BOOL
VAR_INPUT
	jog_activation_condition:	BOOL;
END_VAR
VAR_IN_OUT
    CONVERSION_this:		jog_manager;	(*$ Instance to which the method applies $*)
END_VAR

IF	NOT (descriptor_mode_is_operational(CONVERSION_this.descriptor)
		(*OR
		descriptor_mode_is_test(CONVERSION_this.descriptor)*))	
THEN
	jog_manager_set_jog_activation_condition := FALSE;					(* command rejected *)
 	RETURN;
END_IF

CONVERSION_this.jog_activation_condition := jog_activation_condition;
CONVERSION_this.operational_command := SEL(CONVERSION_this.jog_activation_condition, JOG_MANAGER_RESET_ACTIVATION_CONDITION, JOG_MANAGER_SET_ACTIVATION_CONDITION);
jog_manager_set_jog_activation_condition := TRUE;						(* command accepted *)

END_FUNCTION

// ---- POUs/AFL extensions/jog_manager/commands/jog_manager_set_list_selected.TcPOU
(*$
	Set the jog list selection in <b><i>this</i></b>.
	The method returns <i>TRUE</i> if the command is accepted, otherwise it returns <i>FALSE</i>.
$*)
FUNCTION jog_manager_set_list_selected : BOOL
VAR_INPUT
	list_selected:			UINT;
END_VAR
VAR_IN_OUT
    CONVERSION_this:		jog_manager;	(*$ Instance to which the method applies $*)
END_VAR

IF	NOT (descriptor_mode_is_operational(CONVERSION_this.descriptor)
		(*OR
		descriptor_mode_is_test(CONVERSION_this.descriptor)*))	
THEN
	jog_manager_set_list_selected := FALSE;					(* command rejected *)
 	RETURN;
END_IF

CONVERSION_this.CONVERSION_private.list_selected := list_selected;
jog_manager_set_list_selected := TRUE;						(* command accepted *)

END_FUNCTION

// ---- POUs/AFL extensions/jog_manager/status/jog_manager_is_jog_active.TcPOU
(*$
	Returns <i>TRUE</i> if the status of the instance <b><i>this</i></b> is
	<a href="#jog_manager_status_enum"><i>JOG_MANAGER_STATUS_ACTIVE</i></a>, 
	<i>FALSE</i> otherwise.
$*)
FUNCTION jog_manager_is_jog_active : BOOL
VAR_IN_OUT
    CONVERSION_this:	jog_manager;	(*$ Instance to which the method applies $*)
END_VAR

jog_manager_is_jog_active := (CONVERSION_this.status >= JOG_MANAGER_STATUS_ACTIVE);

END_FUNCTION

// ---- POUs/AFL extensions/jog_manager/commands/jog_manager_stop_jog_absolute_movement.TcPOU
(*$
	Stop the jog absolute movement <b><i>this</i></b>.
	The method returns <i>TRUE</i> if the command is accepted, otherwise it returns <i>FALSE</i>.
$*)
FUNCTION jog_manager_stop_jog_absolute_movement : BOOL
VAR_IN_OUT
    CONVERSION_this:		jog_manager;	(*$ Instance to which the method applies $*)
END_VAR

IF	NOT (descriptor_mode_is_operational(CONVERSION_this.descriptor)
		(*OR
		descriptor_mode_is_test(CONVERSION_this.descriptor)*))	
THEN
	jog_manager_stop_jog_absolute_movement := FALSE;				(* command rejected *)
 	RETURN;
END_IF

CONVERSION_this.operational_command := JOG_MANAGER_STOP_ABSOLUTE_MOVEMENT;
jog_manager_stop_jog_absolute_movement := TRUE;						(* command accepted *)

END_FUNCTION

// ---- POUs/AFL extensions/jog_manager/initialize/jog_manager_init.TcPOU
(*$
	Initializes the instance specified by the parameter <b><i>this</i></b>. <br/>
	<p>
	This function should be called at startup only.<br/>	
	Against errors on the input parameters the cpu is stopped, in this case the cause <br/>
	can be inspected in the global struct <i>framework.abort_error</i>: <br/>
	<br/>
	<li> <b>ERRORID_1 = 1</b>: <b><i>object_name</i></b> is illegal </li>
	</p>
$*)
FUNCTION jog_manager_init : VOID
VAR_INPUT
	object_name:		STRING(MAX_OBJ_NAME_LENGTH);	(*$ The instance name as <i>STRING</i> $*)	
END_VAR
VAR_IN_OUT	
	process:			process;			(*$ <a href="#process_object"><i>process</i></a> membership $*)
	CONVERSION_this:	jog_manager;		(*$ Instance to which the method applies $*)
END_VAR
VAR
	i:					UINT;
END_VAR

IF 	CONVERSION_this.CONVERSION_private.initialized
THEN
	RETURN;
END_IF

IF 	process_is_not_initialized(process)
THEN
	IF 	framework_initialization()
	THEN
		RETURN;
	END_IF
END_IF

IF 	process_is_not_initialized(process)
THEN
	framework_object_not_initialized_get_name(
		object_address := ADR(process), 
		object_size := SIZEOF(process), 
		abort := TRUE,
		error_str_1 := 'object not initialized', 
		error_str_2 := CONCAT('Please check jog_manager_init of ',CONVERSION_this.object_name)			
	);
    RETURN;
END_IF

IF 	object_name = ''
THEN
	framework_object_not_initialized_get_name(
		object_address := ADR(CONVERSION_this), 
		object_size := SIZEOF(CONVERSION_this), 
		abort := TRUE,
		error_str_1 := 'object name is null', 
		error_str_2 := ''
	);
    RETURN;
END_IF

IF 	obj_name_find_illegal_characters(object_name)
THEN
    abort(
		object_name := object_name,
        errorID_1 := 1,
        errorID_2 := 0,
        errorID_3 := 0,
        error_str_1 := CONCAT(CONCAT(CONCAT(CONCAT('(', JOG_MANAGER_CLASS_NAME), ') '), object_name), ' object name is invalid'),
		error_str_2 := ''
    );
    RETURN;
END_IF

CONVERSION_this.object_name := object_name;
CONVERSION_this.CONVERSION_private.my_address := ADR(CONVERSION_this);

descriptor_init(
	object_name := CONCAT(CONVERSION_this.object_name,'.descriptor'),
	process := process,
	CONVERSION_this := CONVERSION_this.descriptor
	);

CONVERSION_this.status := JOG_MANAGER_STATUS_INIT;
CONVERSION_this.command := JOG_MANAGER_CMD_NONE;
CONVERSION_this.test.command := JOG_MANAGER_TEST_CMD_NONE;

FOR i := 1 TO JOG_MANAGER_MAX_PARENTS DO
	CONVERSION_this.parents[i] := G_Framework.NULL;
END_FOR											
CONVERSION_this.parents_next_free := 1;
	
FOR i := JOG_MANAGER_JOG_LIST_NONE TO JOG_MANAGER_JOG_LIST_MAX DO
	CONVERSION_this.axis_list[i].axis := G_framework.NULL;
	CONVERSION_this.axis_list[i].master_axis := FALSE;
	CONVERSION_this.axis_list[i].jog_type := JOG_TYPE_NONE;
	CONVERSION_this.axis_list[i].sw_limit_positive := 0.0;
	CONVERSION_this.axis_list[i].sw_limit_negative := 0.0;
	CONVERSION_this.axis_list[i].all_slave_axis_engaged := FALSE;
END_FOR
CONVERSION_this.CONVERSION_private.list_selected := JOG_MANAGER_JOG_LIST_NONE;

CONVERSION_this.di_pendant_positive := G_framework.NULL;
CONVERSION_this.di_pendant_negative := G_framework.NULL;
CONVERSION_this.has_pendant := FALSE;

CONVERSION_this.has_shared_pendant := G_framework.NULL;
CONVERSION_this.shared_pendant_active := FALSE;

parameter_overwrite_bool_init(
	object_name := CONCAT(CONVERSION_this.object_name, '.jog_active_pow'),
	parameter := CONVERSION_this.jog_active,
	process := process,
	CONVERSION_this := CONVERSION_this.jog_active_pow);

parameter_overwrite_bool_init(
	object_name := CONCAT(CONVERSION_this.object_name, '.enable_sw_limit_pow'),
	parameter := CONVERSION_this.enable_sw_limit,
	process := process,
	CONVERSION_this := CONVERSION_this.enable_sw_limit_pow);

parameter_overwrite_lreal_init(
	object_name := CONCAT(CONVERSION_this.object_name, '.axis_cmd_position_rotative_pow'),
	out_of_range := PARAMETER_OVERWRITE_OUT_OF_RANGE_NONE,
	parameter := CONVERSION_this.axis_cmd_position_rotative,
	process := process,
	CONVERSION_this := CONVERSION_this.axis_cmd_position_rotative_pow);

parameter_overwrite_lreal_init(
	object_name := CONCAT(CONVERSION_this.object_name, '.axis_cmd_position_linear_pow'),
	out_of_range := PARAMETER_OVERWRITE_OUT_OF_RANGE_NONE,
	parameter := CONVERSION_this.axis_cmd_position_linear,
	process := process,
	CONVERSION_this := CONVERSION_this.axis_cmd_position_linear_pow);
			
parameter_overwrite_bool_init(
	object_name := CONCAT(CONVERSION_this.object_name, '.pendant_active_pow'),
	parameter := CONVERSION_this.pendant_active,
	process := process,
	CONVERSION_this := CONVERSION_this.pendant_active_pow);
	
command_button_init(
	object_name := CONCAT(CONVERSION_this.object_name, '.hmi_jog_positive'),
	process := process,
	CONVERSION_this := CONVERSION_this.hmi_jog_positive_cbtn);	

command_button_init(
	object_name := CONCAT(CONVERSION_this.object_name, '.hmi_jog_negative'),
	process := process,
	CONVERSION_this := CONVERSION_this.hmi_jog_negative_cbtn);	

command_button_init(
	object_name := CONCAT(CONVERSION_this.object_name, '.hmi_jog_absolute'),
	process := process,
	CONVERSION_this := CONVERSION_this.hmi_jog_absolute_cbtn);	

hmi_graphic_object_status_init(
	object_name := CONCAT(CONVERSION_this.object_name, '.hmi_jog_selection_hgos'),
	process := process,
	CONVERSION_this  := CONVERSION_this.hmi_jog_selection_hgos);
	
hmi_graphic_object_status_init(
	object_name := CONCAT(CONVERSION_this.object_name, '.hmi_rot_selection_hgos'),
	process := process,
	CONVERSION_this  := CONVERSION_this.hmi_rot_selection_hgos);

hmi_graphic_object_status_init(
	object_name := CONCAT(CONVERSION_this.object_name, '.hmi_lin_selection_hgos'),
	process := process,
	CONVERSION_this  := CONVERSION_this.hmi_lin_selection_hgos);

hmi_graphic_object_status_init(
	object_name := CONCAT(CONVERSION_this.object_name, '.hmi_sw_limit_hgos'),
	process := process,
	CONVERSION_this  := CONVERSION_this.hmi_sw_limit_hgos);

hmi_graphic_object_status_init(
	object_name := CONCAT(CONVERSION_this.object_name, '.hmi_pendant_active_hgos'),
	process := process,
	CONVERSION_this  := CONVERSION_this.hmi_pendant_active_hgos);
	
led_init(
	object_name := CONCAT(CONVERSION_this.object_name, '.hmi_pendant_positive_ld'),
	process := process,
	CONVERSION_this  := CONVERSION_this.hmi_pendant_positive_ld);

led_init(
	object_name := CONCAT(CONVERSION_this.object_name, '.hmi_pendant_negative_ld'),
	process := process,
	CONVERSION_this  := CONVERSION_this.hmi_pendant_negative_ld);
	
CONVERSION_this.CONVERSION_private.initialized := TRUE;

END_FUNCTION

// ---- POUs/AFL extensions/jog_manager/initialize/jog_manager_add_parent.TcPOU
(*$
	Adds the <a href="#jog_manager_object"><i>jog_manager</i></a> that act 
	as parent, to the instance specified by the parameter <i><b>this</i></b>.	
	This function should be called at startup only.<br/>	
	Against errors on the input parameters the cpu is stopped, in this case the cause <br/>
	can be inspected in the global struct <i>framework.abort_error</i>: <br/>
	<br/>
    <li> <b>ERRORID_1 = 9</b>: <b><i>this</i></b> instance parent itself </li>   	
	</p>
$*)
FUNCTION jog_manager_add_parent : BOOL
VAR_IN_OUT
	parent:				jog_manager;	
	CONVERSION_this:	jog_manager;				(*$ Instance to which the method applies $*)
END_VAR
VAR
	i:					UINT;
	found:				BOOL := FALSE;
END_VAR

IF 	jog_manager_is_not_initialized(CONVERSION_this)
   	OR
   	jog_manager_is_not_initialized(parent)
THEN
	IF framework_initialization()
	THEN
		RETURN;
	END_IF
END_IF

IF 	jog_manager_is_not_initialized(CONVERSION_this)
THEN
	framework_object_not_initialized_get_name(
		object_address := ADR(CONVERSION_this),
		object_size := SIZEOF(CONVERSION_this),
		abort := TRUE,
		error_str_1 := 'object not initialized', 
		error_str_2 := CONCAT('Please check jog_manager_init of ', CONVERSION_this.object_name)				
	);
    RETURN;
END_IF

IF 	jog_manager_is_not_initialized(parent)
THEN
	framework_object_not_initialized_get_name(
		object_address := ADR(parent),
		object_size := SIZEOF(parent),
		abort := TRUE,
		error_str_1 := 'object not initialized', 
		error_str_2 := CONCAT('Please check cam_engage_manager_init of ', CONVERSION_this.object_name)				
	);
    RETURN;
END_IF

IF	CONVERSION_this.CONVERSION_private.my_address = ADR(parent)
THEN 
	abort(
		object_name := CONVERSION_this.object_name,
		errorID_1 := 9,
		errorID_2 := 0,
		errorID_3 := 0,
		error_str_1 := CONCAT(CONVERSION_this.object_name, ' jog_manager and parent are equal'),
		error_str_2 := 'jog_manager_add_parent'
		);
	RETURN;
END_IF

IF 	CONVERSION_this.parents_next_free < JOG_MANAGER_MAX_PARENTS
THEN
	FOR i := 1 TO CONVERSION_this.parents_next_free-1 DO
		IF	CONVERSION_this.parents[i] = ADR(parent)
		THEN
			found := TRUE;
			EXIT;
		END_IF
	END_FOR
	IF 	NOT found
	THEN	
		CONVERSION_this.parents[CONVERSION_this.parents_next_free] := ADR(parent);
		CONVERSION_this.parents_next_free := CONVERSION_this.parents_next_free + 1;
	END_IF
	
	jog_manager_add_parent := TRUE;
	RETURN;
end_if
	
jog_manager_add_parent := FALSE;

END_FUNCTION

// ---- POUs/AFL extensions/jog_manager/private/jog_manager_is_not_initialized.TcPOU
(* Function that returns if an object is not initialized. *)
FUNCTION jog_manager_is_not_initialized : BOOL
VAR_IN_OUT
	CONVERSION_this:	jog_manager;	(* object reference *)
END_VAR

jog_manager_is_not_initialized:=NOT CONVERSION_this.CONVERSION_private.initialized;

END_FUNCTION

// ---- POUs/AFL extensions/jog_manager/initialize/jog_manager_add_pendant.TcPOU
(*$
	Adds the <a href="#digital_input_object"><i>digital_input</i></a> that performs 
	the jog plus and jog minus pendant command to the instance specified by the 
	parameter <i><b>this</i></b>.	
	This function should be called at startup only.<br/>	
	Against errors on the input parameters the cpu is stopped, in this case the cause <br/>
	can be inspected in the global struct <i>framework.abort_error</i>: <br/>
	<br/>
    <li> <b>ERRORID_1 = 5</b>: <b><i>this</i></b> instance has already a jog positive digital_input </li>
    <li> <b>ERRORID_1 = 6</b>: <b><i>this</i></b> instance has already a jog negative digital_input </li>		
	</p>
$*)
FUNCTION jog_manager_add_pendant: VOID
VAR_IN_OUT
	di_pendant_positive:	digital_input;
	(*$ Jog positive <a href="#digital_input_object"><i>digital_input</i></a> that has to be added $*)	
	di_pendant_negative:	digital_input;
	(*$ Jog negative <a href="#digital_input_object"><i>digital_input</i></a> that has to be added $*)		
	CONVERSION_this:		jog_manager;	(*$ Instance to which the method applies $*)
END_VAR

IF 	CONVERSION_this.has_pendant
   	AND
   	CONVERSION_this.di_pendant_positive = ADR(di_pendant_positive)
	AND
	CONVERSION_this.di_pendant_negative = ADR(di_pendant_negative)
THEN
	RETURN;
END_IF

IF jog_manager_is_not_initialized(CONVERSION_this)
   OR
   digital_input_is_not_initialized(di_pendant_positive)
   OR
   digital_input_is_not_initialized(di_pendant_negative)
THEN
	IF 	framework_initialization()
	THEN
		RETURN;
	END_IF
END_IF

IF 	jog_manager_is_not_initialized(CONVERSION_this)
THEN
	framework_object_not_initialized_get_name(
		object_address := ADR(CONVERSION_this), 
		object_size := SIZEOF(CONVERSION_this),
		abort := TRUE,
		error_str_1 := 'object not initialized', 
		error_str_2 := 'jog_manager_add_pendant'
	);
    RETURN;
END_IF

IF 	digital_input_is_not_initialized(di_pendant_positive)
THEN
	framework_object_not_initialized_get_name(
		object_address := ADR(di_pendant_positive), 
		object_size := SIZEOF(di_pendant_positive),
		abort := TRUE, 
		error_str_1 := 'object not initialized', 
		error_str_2 := CONCAT('Please check jog_manager_add_pendant of ',CONVERSION_this.object_name)				
	);
    RETURN;
END_IF

IF 	digital_input_is_not_initialized(di_pendant_negative)
THEN
	framework_object_not_initialized_get_name(
		object_address := ADR(di_pendant_negative), 
		object_size := SIZEOF(di_pendant_negative),
		abort := TRUE, 
		error_str_1 := 'object not initialized', 
		error_str_2 := CONCAT('Please check jog_manager_add_pendant of ',CONVERSION_this.object_name)				
	);
    RETURN;
END_IF

IF 	CONVERSION_this.has_pendant
   	AND
   	CONVERSION_this.di_pendant_positive <> ADR(di_pendant_positive)
THEN
    abort(
		object_name := CONVERSION_this.object_name,
        errorID_1 := 5,
        errorID_2 := 0,
        errorID_3 := 0,
        error_str_1 := CONCAT(CONVERSION_this.object_name, ' jog_manager has already a jog positive digital_input'),
		error_str_2 := 'jog_manager_add_pendant'
        );
    RETURN;
END_IF

IF 	CONVERSION_this.has_pendant
   	AND
   	CONVERSION_this.di_pendant_negative <> ADR(di_pendant_negative)
THEN
    abort(
		object_name := CONVERSION_this.object_name,
        errorID_1 := 5,
        errorID_2 := 0,
        errorID_3 := 0,
        error_str_1 := CONCAT(CONVERSION_this.object_name, ' jog_manager has already a jog negative digital_input'),
		error_str_2 := 'jog_manager_add_pendant'
        );
    RETURN;
END_IF

CONVERSION_this.di_pendant_positive := ADR(di_pendant_positive);
CONVERSION_this.di_pendant_negative := ADR(di_pendant_negative);
CONVERSION_this.has_pendant := TRUE;

END_FUNCTION

// ---- POUs/AFL extensions/jog_manager/initialize/jog_manager_add_shared_pendant.TcPOU
(*$
	Adds the reference to <i><b>jog_manager</i></b> that performs 
	the jog plus and jog minus pendant command to the instance specified by the 
	parameter <i><b>this</i></b>.	
	This function should be called at startup only.<br/>	
	Against errors on the input parameters the cpu is stopped, in this case the cause <br/>
	can be inspected in the global struct <i>framework.abort_error</i>: <br/>
	<br/>
    <li> <b>ERRORID_1 = 10</b>: <b><i>this</i></b> instance parent itself  </li>
    <li> <b>ERRORID_1 = 11</b>: <b><i>this</i></b> parent without pendant </li>		
	</p>
$*)
FUNCTION jog_manager_add_shared_pendant : BOOL
VAR_IN_OUT
	parent:				jog_manager;	
	CONVERSION_this:	jog_manager;				(*$ Instance to which the method applies $*)
END_VAR
VAR
	i:					UINT;
	found:				BOOL := FALSE;
END_VAR

IF 	jog_manager_is_not_initialized(CONVERSION_this)
   	OR
   	jog_manager_is_not_initialized(parent)
THEN
	IF framework_initialization()
	THEN
		RETURN;
	END_IF
END_IF

IF 	jog_manager_is_not_initialized(CONVERSION_this)
THEN
	framework_object_not_initialized_get_name(
		object_address := ADR(CONVERSION_this),
		object_size := SIZEOF(CONVERSION_this),
		abort := TRUE,
		error_str_1 := 'object not initialized', 
		error_str_2 := CONCAT('Please check jog_manager_init of ', CONVERSION_this.object_name)				
	);
    RETURN;
END_IF

IF 	jog_manager_is_not_initialized(parent)
THEN
	framework_object_not_initialized_get_name(
		object_address := ADR(parent),
		object_size := SIZEOF(parent),
		abort := TRUE,
		error_str_1 := 'object not initialized', 
		error_str_2 := CONCAT('Please check cam_engage_manager_init of ', CONVERSION_this.object_name)				
	);
    RETURN;
END_IF

IF	CONVERSION_this.CONVERSION_private.my_address = ADR(parent)
THEN 
	abort(
		object_name := CONVERSION_this.object_name,
		errorID_1 := 10,
		errorID_2 := 0,
		errorID_3 := 0,
		error_str_1 := CONCAT(CONVERSION_this.object_name, ' jog_manager and parent are equal'),
		error_str_2 := 'jog_manager_add_shared_pendant'
		);
	RETURN;
END_IF

IF	NOT parent.has_pendant
THEN 
	abort(
		object_name := CONVERSION_this.object_name,
		errorID_1 := 11,
		errorID_2 := 0,
		errorID_3 := 0,
		error_str_1 := CONCAT(CONVERSION_this.object_name, ' jog_manager parent without pendant'),
		error_str_2 := 'jog_manager_add_shared_pendant'
		);
	RETURN;
END_IF

CONVERSION_this.has_shared_pendant := ADR(parent);
jog_manager_add_shared_pendant := TRUE;

END_FUNCTION

// ---- POUs/AFL extensions/jog_manager/jog_manager_cycle.TcPOU
(*$
	Handles the state machine of the object, has to be called once per task cycle <br/>
	<p>
	Against certain errors the cpu can be stopped at the first cycle of the caller task, <br/> 
	in this case the cause can be inspected in the global struct <i>framework.abort_error</i>: <br/>
	<br/>	
$*)
FUNCTION jog_manager_cycle : VOID
VAR_IN_OUT
    CONVERSION_this:	jog_manager;	(*$ Instance to which the method applies $*)
END_VAR
VAR 
	i:					UINT;
END_VAR

IF 	NOT CONVERSION_this.CONVERSION_private.cycle_is_active
THEN
	descriptor_set_task_id(CONVERSION_this.descriptor);

	IF 	jog_manager_is_not_initialized(CONVERSION_this)
	THEN
		framework_object_not_initialized_get_name(
			object_address := ADR(CONVERSION_this),
			object_size := SIZEOF(CONVERSION_this),
			abort := TRUE,
			error_str_1 := 'object not initialized',
			error_str_2 := ''
		);
	    RETURN;
	END_IF

	CONVERSION_this.CONVERSION_private.cycle_is_active := TRUE;
END_IF

IF 	descriptor_mode_req_is_pending(CONVERSION_this.descriptor) 
THEN
    jog_manager_change_mode(CONVERSION_this);
END_IF

command_button_cycle(CONVERSION_this.hmi_jog_positive_cbtn);
command_button_cycle(CONVERSION_this.hmi_jog_negative_cbtn);
command_button_cycle(CONVERSION_this.hmi_jog_absolute_cbtn);

CASE descriptor_get_mode(CONVERSION_this.descriptor) OF
	MODE_ABSENT:
		RETURN;

	MODE_TO_INACTIVE:
		;		(*$FIXME: To inactive mode strategy to handle. $*)

	MODE_INACTIVE:
		;		(*$FIXME: Inactive mode to handle. $*)

	MODE_TEST:
		CONVERSION_this.command := jog_manager_test_command_handler(CONVERSION_this);

	MODE_OPERATIONAL:
		CONVERSION_this.command := CONVERSION_this.operational_command;

END_CASE;

jog_manager_read_inputs(CONVERSION_this);
jog_manager_submit_command(CONVERSION_this);

(*Selection validation*)
CONVERSION_this.CONVERSION_private.old_list_selected_is_valid :=
	(CONVERSION_this.CONVERSION_private.old_list_selected > JOG_MANAGER_JOG_LIST_NONE)
	AND
	(CONVERSION_this.CONVERSION_private.old_list_selected <= JOG_MANAGER_JOG_LIST_MAX);
IF	CONVERSION_this.CONVERSION_private.old_list_selected_is_valid
THEN	
	CONVERSION_this.CONVERSION_private.old_list_selected_axis_is_valid := CONVERSION_this.axis_list[CONVERSION_this.CONVERSION_private.old_list_selected].axis <> G_framework.NULL;
ELSE
	CONVERSION_this.CONVERSION_private.old_list_selected_axis_is_valid := FALSE;
END_IF
IF 	CONVERSION_this.CONVERSION_private.update_parameters > 0
THEN
	CONVERSION_this.CONVERSION_private.update_parameters := CONVERSION_this.CONVERSION_private.update_parameters + 1;
END_IF
	
(*Old selection validation*)
CONVERSION_this.CONVERSION_private.list_selected_is_valid :=
	(CONVERSION_this.CONVERSION_private.list_selected > JOG_MANAGER_JOG_LIST_NONE)
	AND
	(CONVERSION_this.CONVERSION_private.list_selected <= JOG_MANAGER_JOG_LIST_MAX);
IF	CONVERSION_this.CONVERSION_private.list_selected_is_valid
THEN
	CONVERSION_this.CONVERSION_private.list_selected_axis_is_valid := CONVERSION_this.axis_list[CONVERSION_this.CONVERSION_private.list_selected].axis <> G_framework.NULL;
ELSE
	CONVERSION_this.CONVERSION_private.list_selected_axis_is_valid := FALSE;
END_IF
 
(*SW limit and jog direction management*)
IF 	CONVERSION_this.CONVERSION_private.list_selected_axis_is_valid
THEN		
	CONVERSION_this.CONVERSION_private.sw_limit_active :=
		(axis_get_modulo(CONVERSION_this.axis_list[CONVERSION_this.CONVERSION_private.list_selected].axis^) = 0.0)
		AND
		(
			(ABS(CONVERSION_this.axis_list[CONVERSION_this.CONVERSION_private.list_selected].sw_limit_negative) > 0.0)
			OR
			(ABS(CONVERSION_this.axis_list[CONVERSION_this.CONVERSION_private.list_selected].sw_limit_positive) > 0.0)
		);

	CONVERSION_this.CONVERSION_private.axis_is_linear := 
		(CONVERSION_this.axis_list[CONVERSION_this.CONVERSION_private.list_selected].jog_type = JOG_TYPE_LINEAR)
		OR
		(CONVERSION_this.axis_list[CONVERSION_this.CONVERSION_private.list_selected].jog_type = JOG_TYPE_LINEAR_PLUS)
		OR
		(CONVERSION_this.axis_list[CONVERSION_this.CONVERSION_private.list_selected].jog_type = JOG_TYPE_LINEAR_MINUS);
		
	CONVERSION_this.CONVERSION_private.axis_is_rotative := 
		(CONVERSION_this.axis_list[CONVERSION_this.CONVERSION_private.list_selected].jog_type = JOG_TYPE_ROTATIVE)
		OR
		(CONVERSION_this.axis_list[CONVERSION_this.CONVERSION_private.list_selected].jog_type = JOG_TYPE_ROTATIVE_PLUS)
		OR
		(CONVERSION_this.axis_list[CONVERSION_this.CONVERSION_private.list_selected].jog_type = JOG_TYPE_ROTATIVE_MINUS);
		
	CONVERSION_this.CONVERSION_private.jog_positive_enable :=
		(CONVERSION_this.axis_list[CONVERSION_this.CONVERSION_private.list_selected].jog_type = JOG_TYPE_LINEAR)
		OR
		(CONVERSION_this.axis_list[CONVERSION_this.CONVERSION_private.list_selected].jog_type = JOG_TYPE_LINEAR_PLUS)
		OR	
		(CONVERSION_this.axis_list[CONVERSION_this.CONVERSION_private.list_selected].jog_type = JOG_TYPE_ROTATIVE)
		OR
		(CONVERSION_this.axis_list[CONVERSION_this.CONVERSION_private.list_selected].jog_type = JOG_TYPE_ROTATIVE_PLUS);	
	
	CONVERSION_this.CONVERSION_private.jog_negative_enable :=
		(CONVERSION_this.axis_list[CONVERSION_this.CONVERSION_private.list_selected].jog_type = JOG_TYPE_LINEAR)
		OR
		(CONVERSION_this.axis_list[CONVERSION_this.CONVERSION_private.list_selected].jog_type = JOG_TYPE_LINEAR_MINUS)
		OR	
		(CONVERSION_this.axis_list[CONVERSION_this.CONVERSION_private.list_selected].jog_type = JOG_TYPE_ROTATIVE)
		OR
		(CONVERSION_this.axis_list[CONVERSION_this.CONVERSION_private.list_selected].jog_type = JOG_TYPE_ROTATIVE_MINUS);	
		
	CONVERSION_this.CONVERSION_private.sw_limit_active_positive :=
		CONVERSION_this.CONVERSION_private.sw_limit_active
		AND
		CONVERSION_this.enable_sw_limit
		AND
		(
			(
				CONVERSION_this.CONVERSION_private.axis_is_linear
				AND
				(CONVERSION_this.axis_act_position_linear >= CONVERSION_this.axis_list[CONVERSION_this.CONVERSION_private.list_selected].sw_limit_positive)
			)
			OR
			(
				CONVERSION_this.CONVERSION_private.axis_is_rotative
				AND
				(CONVERSION_this.axis_act_position_rotative >= CONVERSION_this.axis_list[CONVERSION_this.CONVERSION_private.list_selected].sw_limit_positive)
			)
		);
		
	CONVERSION_this.CONVERSION_private.sw_limit_active_negative :=
		CONVERSION_this.CONVERSION_private.sw_limit_active
		AND
		CONVERSION_this.enable_sw_limit
		AND
		(
			(
				CONVERSION_this.CONVERSION_private.axis_is_linear
				AND
				(CONVERSION_this.axis_act_position_linear <= CONVERSION_this.axis_list[CONVERSION_this.CONVERSION_private.list_selected].sw_limit_negative)
			)
			OR
			(
				CONVERSION_this.CONVERSION_private.axis_is_rotative
				AND
				(CONVERSION_this.axis_act_position_rotative <= CONVERSION_this.axis_list[CONVERSION_this.CONVERSION_private.list_selected].sw_limit_negative)
			)
		);			
ELSE
	CONVERSION_this.CONVERSION_private.sw_limit_active := FALSE;
	CONVERSION_this.CONVERSION_private.axis_is_linear := FALSE;
	CONVERSION_this.CONVERSION_private.axis_is_rotative := FALSE;
END_IF
	
(*Transition states*)
CASE CONVERSION_this.status OF
	
	JOG_MANAGER_STATUS_INIT:
		parameter_overwrite_set_bool_value(FALSE, CONVERSION_this.jog_active_pow);
		parameter_overwrite_set_bool_value(FALSE, CONVERSION_this.pendant_active_pow);
		CONVERSION_this.CONVERSION_private.update_parameters := 0;		
    	CONVERSION_this.status := JOG_MANAGER_STATUS_IDLE;

    JOG_MANAGER_STATUS_IDLE:
		;
		
    JOG_MANAGER_STATUS_READY:
        IF	CONVERSION_this.jog_active
		THEN		
			FOR i := 1 TO CONVERSION_this.parents_next_free-1 DO
				IF	CONVERSION_this.parents[i]^.jog_active
				THEN
					parameter_overwrite_set_bool_value(FALSE, CONVERSION_this.parents[i]^.jog_active_pow);
				END_IF	
			END_FOR
			CONVERSION_this.CONVERSION_private.old_list_selected := JOG_MANAGER_JOG_LIST_NONE;			
			CONVERSION_this.status := JOG_MANAGER_STATUS_ACTIVE;
		END_IF
    
	JOG_MANAGER_STATUS_ACTIVE:
        IF	NOT CONVERSION_this.jog_active
		THEN
			IF	CONVERSION_this.CONVERSION_private.list_selected_axis_is_valid					 
			THEN
				IF	axis_is_disabled(CONVERSION_this.axis_list[CONVERSION_this.CONVERSION_private.list_selected].axis^)
				THEN
					CONVERSION_this.status := JOG_MANAGER_STATUS_READY;
				ELSE					
					CONVERSION_this.status := JOG_MANAGER_STATUS_SEL_DISABLE_AXIS;										
				END_IF
			ELSE
				CONVERSION_this.status := JOG_MANAGER_STATUS_READY;
			END_IF
		END_IF
		
		IF 	CONVERSION_this.CONVERSION_private.list_selected <> CONVERSION_this.CONVERSION_private.old_list_selected
		THEN					
			CONVERSION_this.CONVERSION_private.update_parameters := 1;							
			IF	CONVERSION_this.CONVERSION_private.old_list_selected_axis_is_valid					 
			THEN								
				CONVERSION_this.status := JOG_MANAGER_STATUS_OLD_DISABLE_AXIS;	
			ELSE
				CONVERSION_this.CONVERSION_private.old_list_selected := CONVERSION_this.CONVERSION_private.list_selected;							
			END_IF				
		ELSIF CONVERSION_this.CONVERSION_private.list_selected_axis_is_valid
		THEN
			IF 	axis_is_disabled(CONVERSION_this.axis_list[CONVERSION_this.CONVERSION_private.list_selected].axis^)
				AND
				axis_is_ok(FALSE, CONVERSION_this.axis_list[CONVERSION_this.CONVERSION_private.list_selected].axis^)
				AND
				(
					NOT CONVERSION_this.axis_list[CONVERSION_this.CONVERSION_private.list_selected].master_axis
					OR
					CONVERSION_this.axis_list[CONVERSION_this.CONVERSION_private.list_selected].all_slave_axis_engaged
				)
			THEN
				CONVERSION_this.status := JOG_MANAGER_STATUS_SEL_ENABLE_AXIS;
			END_IF
		END_IF
    
	JOG_MANAGER_STATUS_SEL_DISABLE_AXIS:
		axis_disable(CONVERSION_this.axis_list[CONVERSION_this.CONVERSION_private.list_selected].axis^);
		IF	axis_is_disabled(CONVERSION_this.axis_list[CONVERSION_this.CONVERSION_private.list_selected].axis^)
		THEN									
			CONVERSION_this.status := JOG_MANAGER_STATUS_READY;			
		END_IF
		
	JOG_MANAGER_STATUS_OLD_DISABLE_AXIS:
		axis_disable(CONVERSION_this.axis_list[CONVERSION_this.CONVERSION_private.old_list_selected].axis^);
		IF	axis_is_disabled(CONVERSION_this.axis_list[CONVERSION_this.CONVERSION_private.old_list_selected].axis^)
		THEN	
			CONVERSION_this.CONVERSION_private.old_list_selected := CONVERSION_this.CONVERSION_private.list_selected;		
			CONVERSION_this.status := JOG_MANAGER_STATUS_ACTIVE;			
		END_IF
	
	JOG_MANAGER_STATUS_SEL_ENABLE_AXIS:
		axis_enable(CONVERSION_this.axis_list[CONVERSION_this.CONVERSION_private.list_selected].axis^);
		IF	axis_is_standstill(CONVERSION_this.axis_list[CONVERSION_this.CONVERSION_private.list_selected].axis^)
		THEN						
			CONVERSION_this.status := JOG_MANAGER_STATUS_SEL_ENABLED_AXIS;			
		END_IF
		
	JOG_MANAGER_STATUS_SEL_ENABLED_AXIS:
		IF	NOT CONVERSION_this.jog_active
			OR
			(CONVERSION_this.CONVERSION_private.list_selected <> CONVERSION_this.CONVERSION_private.old_list_selected)
		THEN
			CONVERSION_this.status := JOG_MANAGER_STATUS_ACTIVE;
		END_IF
		
		(*Jog positive linear*)
		IF 	(
				command_button_is_pressed(CONVERSION_this.hmi_jog_positive_cbtn)
				OR
				(
					CONVERSION_this.has_pendant
					AND
					CONVERSION_this.pendant_active
					AND
					CONVERSION_this.CONVERSION_private.jog_positive_enable
					AND
					NOT CONVERSION_this.CONVERSION_private.sw_limit_active_positive
					AND
					CONVERSION_this.CONVERSION_private.jog_pendant_positive
				)
				OR
				(
					(CONVERSION_this.has_shared_pendant <> G_framework.NULL)
					AND
					CONVERSION_this.shared_pendant_active 
					AND
					CONVERSION_this.CONVERSION_private.jog_positive_enable
					AND
					NOT CONVERSION_this.CONVERSION_private.sw_limit_active_positive
					AND
					CONVERSION_this.CONVERSION_private.jog_pendant_positive
				)
			)
			AND 
			(
				(CONVERSION_this.axis_list[CONVERSION_this.CONVERSION_private.list_selected].jog_type = JOG_TYPE_LINEAR)
				OR
				(CONVERSION_this.axis_list[CONVERSION_this.CONVERSION_private.list_selected].jog_type = JOG_TYPE_LINEAR_PLUS)				
			) 
			AND
			(CONVERSION_this.axis_speed_linear > 0.0)
		THEN
			axis_move_velocity(
				velocity			:= MIN(CONVERSION_this.axis_speed_linear, CONVERSION_this.axis_list[CONVERSION_this.CONVERSION_private.list_selected].axis^.parameters.max_velocity),
				acceleration		:= CONVERSION_this.axis_list[CONVERSION_this.CONVERSION_private.list_selected].axis^.parameters.max_acceleration/csp_main_jogManager.AccDec_divider,
				deceleration		:= CONVERSION_this.axis_list[CONVERSION_this.CONVERSION_private.list_selected].axis^.parameters.max_deceleration/csp_main_jogManager.AccDec_divider,
				jerk				:= CONVERSION_this.axis_list[CONVERSION_this.CONVERSION_private.list_selected].axis^.parameters.max_jerk/csp_main_jogManager.AccDec_divider,
				buffer_mode			:= AXIS_BUFFER_MODE_BUFFERED,
				CONVERSION_this		:= CONVERSION_this.axis_list[CONVERSION_this.CONVERSION_private.list_selected].axis^);
			CONVERSION_this.status := JOG_MANAGER_STATUS_LINEAR_JOG_POSITIVE;
		END_IF
		
		(*Jog negative linear*)
		IF	(
				command_button_is_pressed(CONVERSION_this.hmi_jog_negative_cbtn)
				OR
				(
					CONVERSION_this.has_pendant
					AND
					CONVERSION_this.pendant_active
					AND
					CONVERSION_this.CONVERSION_private.jog_negative_enable
					AND
					NOT CONVERSION_this.CONVERSION_private.sw_limit_active_negative
					AND
					CONVERSION_this.CONVERSION_private.jog_pendant_negative
				)
				OR
				(
					(CONVERSION_this.has_shared_pendant <> G_framework.NULL)
					AND
					CONVERSION_this.shared_pendant_active
					AND
					CONVERSION_this.CONVERSION_private.jog_negative_enable
					AND
					NOT CONVERSION_this.CONVERSION_private.sw_limit_active_negative
					AND
					CONVERSION_this.CONVERSION_private.jog_pendant_negative
				)
			)
			AND 
			(
				(CONVERSION_this.axis_list[CONVERSION_this.CONVERSION_private.list_selected].jog_type = JOG_TYPE_LINEAR)
				OR
				(CONVERSION_this.axis_list[CONVERSION_this.CONVERSION_private.list_selected].jog_type = JOG_TYPE_LINEAR_MINUS)				
			) 
			AND
			(CONVERSION_this.axis_speed_linear > 0.0)
		THEN
			axis_move_velocity(
				velocity			:= MAX(-CONVERSION_this.axis_speed_linear, -CONVERSION_this.axis_list[CONVERSION_this.CONVERSION_private.list_selected].axis^.parameters.max_velocity),
				acceleration		:= CONVERSION_this.axis_list[CONVERSION_this.CONVERSION_private.list_selected].axis^.parameters.max_acceleration/csp_main_jogManager.AccDec_divider,
				deceleration		:= CONVERSION_this.axis_list[CONVERSION_this.CONVERSION_private.list_selected].axis^.parameters.max_deceleration/csp_main_jogManager.AccDec_divider,
				jerk				:= CONVERSION_this.axis_list[CONVERSION_this.CONVERSION_private.list_selected].axis^.parameters.max_jerk/csp_main_jogManager.AccDec_divider,
				buffer_mode			:= AXIS_BUFFER_MODE_BUFFERED,
				CONVERSION_this		:= CONVERSION_this.axis_list[CONVERSION_this.CONVERSION_private.list_selected].axis^);
			CONVERSION_this.status := JOG_MANAGER_STATUS_LINEAR_JOG_NEGATIVE;
		END_IF
		
